// TIA Portal V17 program export: 1 tag tables, 1 data types, 3 data blocks, 11 code blocks (in call order from the OBs), 12 instance data blocks

VAR_GLOBAL   // PLC tag table "Default tag table"
   System_Byte AT %MB1 : Byte;
   FirstScan AT %M1.0 : Bool;
   DiagStatusUpdate AT %M1.1 : Bool;
   AlwaysTRUE AT %M1.2 : Bool;
   AlwaysFALSE AT %M1.3 : Bool;
   Clock_Byte AT %MB0 : Byte;
   Clock_10Hz AT %M0.0 : Bool;
   Clock_5Hz AT %M0.1 : Bool;
   "Clock_2.5Hz" AT %M0.2 : Bool;
   Clock_2Hz AT %M0.3 : Bool;
   "Clock_1.25Hz" AT %M0.4 : Bool;
   Clock_1Hz AT %M0.5 : Bool;
   "Clock_0.625Hz" AT %M0.6 : Bool;
   "Clock_0.5Hz" AT %M0.7 : Bool;
   MR_Pulse AT %Q4.0 : Bool;
   MA_Pulse AT %Q4.1 : Bool;
   MR_Direction AT %Q0.0 : Bool;
   MRenable AT %M2.0 : Bool;
   MRReset AT %M2.1 : Bool;
   MRHalt AT %M2.2 : Bool;
   "MRJog-" AT %M2.3 : Bool;
   "MRJog+" AT %M2.4 : Bool;
   MRMoveRelative AT %M2.5 : Bool;
   MRMoveAbsolute AT %M2.6 : Bool;
   MA_Direction AT %Q0.1 : Bool;
   MRPower AT %M2.7 : Bool;
   MRVelocity AT %M3.0 : Bool;
   MREnabled AT %M3.5 : Bool;
   MRHomed AT %M3.1 : Bool;
   MRMoveAbsDone AT %M3.2 : Bool;
   MRStandstill AT %M3.3 : Bool;
   MRError AT %M3.4 : Bool;
   MRActualVelocity AT %MD4 : Real;
   MRActualPosition AT %MD8 : Real;
   MS_Direction AT %Q0.2 : Bool;
   ME_Direction AT %Q0.3 : Bool;
   MS_Pulse AT %Q4.2 : Bool;
   ME_Pulse AT %Q4.3 : Bool;
   AUTOMATICO AT %M3.6 : Bool;
   MANUALE AT %M3.7 : Bool;
   RIPRISTINO AT %M12.0 : Bool;
   PASSO_RIP_01 AT %M12.1 : Bool;
   PASSO_RIP_02 AT %M12.2 : Bool;
   PASSO_RIP_03 AT %M12.3 : Bool;
   STARTCICLO AT %M12.6 : Bool;
   PASSO_CICLO_01 AT %M12.7 : Bool;
   PASSO_CICLO_03 AT %M13.0 : Bool;
   PASSO_CICLO_02 AT %M13.1 : Bool;
   MRSpQuotaMoveRel AT %MD14 : Real;
   MRSpVelocitaMoveRel AT %MD18 : Real;
   MRSpQuotaMoveAbs AT %MD22 : Real;
   MRSpVelocitaMoveAbs AT %MD26 : Real;
   AUX_OK AT %M12.4 : Bool;
   AUX_OK_T AT %M12.5 : Bool;
   RESET_ALLARMI AT %M13.2 : Bool;
   MR_MAN_RELATIVE AT %M13.3 : Bool;
   MR_MAN_ABSOLUTE AT %M13.4 : Bool;
   MR_MAN_HALT AT %M13.5 : Bool;
   MS_MAN_HALT AT %M13.6 : Bool;
   MS_MAN_RELATIVE AT %M13.7 : Bool;
   MS_MAN_ABSOLUTE AT %M30.0 : Bool;
   MA_MAN_HALT AT %M30.1 : Bool;
   MA_MAN_RELATIVE AT %M30.2 : Bool;
   MA_MAN_ABSOLUTE AT %M30.3 : Bool;
   ME_MAN_HALT AT %M30.4 : Bool;
   ME_MAN_RELATIVE AT %M30.5 : Bool;
   ME_MAN_ABSOLUTE AT %M30.6 : Bool;
   "E0.0 FC HOMING MS" AT %I0.0 : Bool;
   ALLA_01_FC_HOMING_MS AT %M30.7 : Bool;
   PASSO_PASSO AT %M31.0 : Bool;
   RIPRISTINATO AT %M31.1 : Bool;
   "E0.1 FC HOMING MR" AT %I0.1 : Bool;
   ALLA_02_FC_HOMING_MR AT %M31.2 : Bool;
END_VAR

TYPE "UDTMotori"
// stored: IsFailsafeCompliant false
   STRUCT
      pos : Struct
         "1" : Real;
         "2" : Real;
         "3" : Real;
         "4" : Real;
         "5" : Real;
      END_STRUCT;
      vel : Struct
         "1" : Real;
         "2" : Real;
         "3" : Real;
         "4" : Real;
         "5" : Real;
      END_STRUCT;
      acc : Struct
         "1" : Real;
         "2" : Real;
         "3" : Real;
         "4" : Real;
         "5" : Real;
      END_STRUCT;
      dec : Struct
         "1" : Real;
         "2" : Real;
         "3" : Real;
         "4" : Real;
         "5" : Real;
      END_STRUCT;
      IN : Struct
         Exe_MC_Reset : Bool;   // comando di reset
         En_MC_Power : Bool;   // abilitazione asse
         Exe_MC_Home : Bool;   // comando di homing
         Sp_Offset_Homing : Real;   // offset azzeramento
         Exe_MC_Halt : Bool;   // comando HALT
         Exe_Jog_Fwd : Bool;   // comando jog +
         Exe_Jog_Bkw : Bool;   // comando jog -
         Sp_Jog_Velocity : Real;   // set velocità JOG
         Exe_MC_Velocity : Bool;   // comando velocità
         Sp_MC_Velocity : Real;   // set velocità Move Velocity
         Exe_MC_MoveRelative : Bool;   // comando posizione relativa
         Sp_MoveRel_Distance : Real;   // set distanza Move Relative
         Sp_MoveRel_Velocity : Real;   // set velocità Move Relative
         Exe_MC_MoveAbs : Bool;   // comando posizione assoluta
         Sp_MoveAbs_Position : Real;   // set posizione Move Absolute
         Sp_MoveAbs_Velocity : Real;   // set velocità Move Absolute
         Exe_MC_ChangeDyna : Bool;   // comando cambio dinamica
         Sp_RampUpTime : Real;   // set tempo di rampa acc [s]
         Sp_RampDnTime : Real;   // set tempo di rampa dec [s]
      END_STRUCT;
      OUT : Struct
         Output_MC_Reset_Done : Bool;   // asse resettato
         Output_MC_AxisEnabled : Bool;   // asse abilitato
         Output_MC_AxisHomed : Bool;   // asse homed (referenziato)
         Output_MC_Halt_Done : Bool;   // asse in halt
         Output_MC_JogInVelocity : Bool;   // vel raggiunta
         Output_MC_MoveInVelocity : Bool;   // vel raggiunta
         Output_MC_MoveRel_Done : Bool;   // move realtive eseguito
         Output_MC_MoveAbs_Done : Bool;   // move absolute eseguito
         Output_MC_MoveAbs_Busy : Bool;   // move absolute in corso
         Output_MC_At_Standstill : Bool;   // asse fermo
         Output_MC_Error : Bool;   // asse in errore (or di vari bool)
         Output_ActVelocity : Real;   // velocity attuale (asse)
         Output_ActPos : Real;   // posizione attuale
      END_STRUCT;
   END_STRUCT;
END_TYPE

DATA_BLOCK "RICETTE"   // DB18
{ S7_Optimized_Access := 'TRUE' }
VERSION : 0.1
// stored: AutoNumber true, DBAccessibleFromOPCUA true, IsOnlyStoredInLoadMemory false, IsRetainMemResEnabled false, IsWriteProtectedInAS false, MemoryReserve 100
   VAR
      nomeRicetta : WString;
   END_VAR
BEGIN
END_DATA_BLOCK

DATA_BLOCK "DBParAssi"   // DB12
{ S7_Optimized_Access := 'TRUE' }
VERSION : 0.1
// stored: AutoNumber true, DBAccessibleFromOPCUA true, IsOnlyStoredInLoadMemory false, IsRetainMemResEnabled false, IsWriteProtectedInAS false, MemoryReserve 100
   VAR RETAIN
      MR : "UDTMotori";
      MA { S7_SetPoint := 'True'} : "UDTMotori";
      MS { S7_SetPoint := 'True'} : "UDTMotori";
      ME { S7_SetPoint := 'True'} : "UDTMotori";
   END_VAR
BEGIN
   MR.pos."1" := 120.0;   // [°] predisposizione (detorsione)
   MR.pos."2" := 10.0;   // [°] quota intermedia (detorsione parziale) / [°] quota intermedia
   MR.pos."3" := 0.0;   // [°] zero / [°]
   MR.pos."4" := 180.0;   // [°] ritorsione
   MR.vel."1" := 1000.0;   // [°/s] vel detorsione
   MR.vel."2" := 1000.0;   // [°/s] vel detorsione parziale
   MR.vel."3" := 200.0;   // [°/s] vel
   MR.vel."4" := 200.0;   // [°/s] vel ritorsione
   MR.IN.Sp_Jog_Velocity := 80.0;
   MR.IN.Sp_MoveRel_Velocity := 1000.0;
   MR.IN.Sp_MoveAbs_Velocity := 1000.0;
   MR.IN.Sp_RampUpTime := 2.0;
   MR.IN.Sp_RampDnTime := 2.0;
   MA.pos."1" := 7.5;   // [mm] quota detorsione / [mm]
   MA.pos."2" := 12.5;   // [mm] quota fissa era 12.5 / [mm]
   MA.pos."3" := 9.6;   // [mm] quota ritorsione / [mm]
   MA.pos."4" := 0.0;   // [mm]
   MA.IN.Sp_Jog_Velocity := 5.0;
   MA.IN.Sp_MoveRel_Velocity := 150.0;
   MA.IN.Sp_MoveAbs_Velocity := 50.0;
   MS.pos."1" := 220.0;   // [pulses] preset (800 0 giro completo) / [pulses] preset (400 0 giro completo)
   // MS.pos."2" : [pulses]
   MS.pos."3" := 95.0;   // [p] quota MA
   MS.vel."1" := 3000.0;   // [p/s]
   MS.vel."3" := 3000.0;   // [p/s]
   MS.IN.Sp_Jog_Velocity := 180.0;
   MS.IN.Sp_MoveRel_Distance := 230.0;
   MS.IN.Sp_MoveRel_Velocity := 1000.0;
   MS.IN.Sp_MoveAbs_Velocity := 1000.0;
   ME.pos."1" := 120.0;   // [°] quota blocco fili / [°]
   ME.pos."2" := 0.0;   // [°] Home position / [°]
   ME.IN.Sp_Jog_Velocity := 200.0;
   ME.IN.Sp_MoveRel_Velocity := 1000.0;
   ME.IN.Sp_MoveAbs_Velocity := 1000.0;
END_DATA_BLOCK

DATA_BLOCK "DB_ALLA"   // DB1
{ S7_Optimized_Access := 'FALSE' }
VERSION : 0.1
// stored: AutoNumber true, DBAccessibleFromOPCUA true, IsOnlyStoredInLoadMemory false, IsWriteProtectedInAS false
   VAR
      wordAlla01 : Word;
   END_VAR
BEGIN
END_DATA_BLOCK

ORGANIZATION_BLOCK "Main"   // OB1, LAD, ProgramCycle
TITLE = "Main Program Sweep (Cycle)"
{ S7_Optimized_Access := 'TRUE' }
VERSION : 0.1
// stored: AutoNumber true, IsIECCheckEnabled false, SetENOAutomatically false
   VAR_INPUT
      Initial_Call : Bool;   // Initial call of this OB
      Remanence : Bool;   // =True, if remanent data are available
   END_VAR
BEGIN

REGION Network 1 (SCL): FORZAMENTI

   //"E0.0 FC HOMING MS" := TRUE;
END_REGION

REGION Network 2 (SCL): LANCIO BLOCCHI

   "RESET_GENERALE"("FirstScan");
   "RESET_ALLA"("RESET_ALLARMI");


   "FB_STATI_MACCHINA_DB"();

   // CICLI
   "FB_RIPRISTINO_GEN_DB"();

   "FB_RIPRISTINO_MR_DB"();
   "FB_RIPRISTINO_MA_DB"();
   "FB_RIPRISTINO_MS_DB"();
   "FB_RIPRISTINO_ME_DB"();

   "FB_CICLO_DB"();

   "FB_ORG_ASSI_DB"();

   "ALLARMI_DB"();
END_REGION
END_ORGANIZATION_BLOCK

FUNCTION_BLOCK "FB_STATI_MACCHINA"   // FB2, LAD
{ S7_Optimized_Access := 'TRUE' }
VERSION : 0.1
// stored: AutoNumber true, IsIECCheckEnabled false, IsRetainMemResEnabled false, MemoryReserve 100, SetENOAutomatically false, UDAEnableTagReadback false
   VAR
      TAux { S7_SetPoint := 'True'} : TON_TIME;
      TResetAlla { S7_SetPoint := 'True'} : TON_TIME;
   END_VAR
BEGIN

REGION Network 1: AUX OK
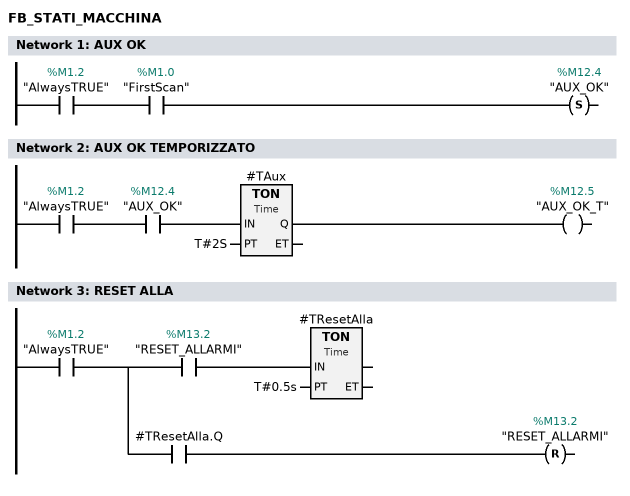
   RUNG wire#powerrail
      Contact( "AlwaysTRUE" )
      Contact( "FirstScan" )
      S_Coil( "AUX_OK" )
   END_RUNG
   // the same network as SCL:
   IF "AlwaysTRUE" AND "FirstScan" THEN "AUX_OK" := TRUE; END_IF;
END_REGION

REGION Network 2: AUX OK TEMPORIZZATO
   RUNG wire#powerrail
      Contact( "AlwaysTRUE" )
      Contact( "AUX_OK" )
      { S7_Templates := "time_type := Time" } #TAux.TON(pt := T#2S, et =>)
      Coil( "AUX_OK_T" )
   END_RUNG
   // the same network as SCL:
   #TAux(IN := "AlwaysTRUE" AND "AUX_OK", PT := T#2S);   // TON
   "AUX_OK_T" := #TAux.Q;
END_REGION

REGION Network 3: RESET ALLA
   RUNG wire#powerrail
      Contact( "AlwaysTRUE" )
      wire#w1
      Contact( "RESET_ALLARMI" )
      { S7_Templates := "time_type := Time" } #TResetAlla.TON(pt := T#0.5s, et =>)
   END_RUNG
   RUNG wire#w1
      Contact( #TResetAlla.Q )
      R_Coil( "RESET_ALLARMI" )
   END_RUNG
   // the same network as SCL:
   #TResetAlla(IN := "AlwaysTRUE" AND "RESET_ALLARMI", PT := T#0.5s);   // TON
   IF "AlwaysTRUE" AND #TResetAlla.Q THEN "RESET_ALLARMI" := FALSE; END_IF;
END_REGION

REGION Network 4 (SCL): MAN/AUTO

   "MANUALE" := NOT "AUTOMATICO";
END_REGION
END_FUNCTION_BLOCK

FUNCTION_BLOCK "FB_RIPRISTINO_GEN"
{ S7_Optimized_Access := 'TRUE' }
VERSION : 0.1
   VAR_OUTPUT 
      bDone : Bool;   // bDone
      fase : Int := 0;   // fase attiva
   END_VAR

   VAR_IN_OUT 
      bStart : Bool;   // start ciclo
   END_VAR

   VAR 
      condOkRipristino : Bool;
      T10 {InstructionName := 'TON_TIME'; LibVersion := '1.0'; S7_SetPoint := 'False'} : TON_TIME;
      T20 {InstructionName := 'TON_TIME'; LibVersion := '1.0'} : TON_TIME;
   END_VAR


BEGIN
	// ripristino generale
	
	#T10(IN := #fase = 10,
	     PT := t#1s);
	
	#T20(IN := #fase = 20,
	     PT := t#1s);
	
	// CONDIZIONI 
	// 
	#condOkRipristino := NOT "STARTCICLO" AND "AUX_OK_T";
	
	// reset start
	// 
	IF NOT #condOkRipristino THEN
	    "RIPRISTINO" := FALSE;
	END_IF;
	
	
	CASE #fase OF
	        
	    0: // attesa start ciclo
	        IF "RIPRISTINO" AND #condOkRipristino THEN
	            // comandi
	            // 
	            "FB_RIPRISTINO_MR_DB".bDone := FALSE;
	            "FB_RIPRISTINO_MA_DB".bDone := FALSE;
	            "FB_RIPRISTINO_MS_DB".bDone := FALSE;
	            "FB_RIPRISTINO_ME_DB".bDone := FALSE;
	            "RIPRISTINATO" := FALSE;
	            
	            "FB_RIPRISTINO_MA_DB".bStart := TRUE;
	            "FB_RIPRISTINO_ME_DB".bStart := TRUE;
	            
	            #fase := 10;
	        END_IF;
	        
	    10:
	        IF "FB_RIPRISTINO_MA_DB".bDone AND "FB_RIPRISTINO_ME_DB".bDone
	        THEN
	            // comandi 
	            // 
	            "FB_RIPRISTINO_MR_DB".bStart := TRUE;
	            "FB_RIPRISTINO_MS_DB".bStart := TRUE;
	            
	            #fase := 30;
	        END_IF;
	        
	    30: // fineciclo
	        IF   "FB_RIPRISTINO_MR_DB".bDone AND   "FB_RIPRISTINO_MS_DB".bDone        THEN
	            // comandi 
	            "RIPRISTINO" := FALSE;
	            "RIPRISTINATO" := TRUE;
	            #bDone := TRUE;
	            
	            #fase := 0;
	        END_IF;
	        
	END_CASE;
	
	
END_FUNCTION_BLOCK

FUNCTION_BLOCK "FB_ORG_ASSI"   // FB5, LAD
{ S7_Optimized_Access := 'TRUE' }
VERSION : 0.1
// stored: AutoNumber true, IsIECCheckEnabled false, IsRetainMemResEnabled false, MemoryReserve 100, SetENOAutomatically false, UDAEnableTagReadback false
   VAR
      CTRL_ASSE_STD_MA { S7_SetPoint := 'True'} : "CTRL_ASSE_STD";
      CTRL_ASSE_STD_MR { S7_SetPoint := 'True'} : "CTRL_ASSE_STD";
      CTRL_ASSE_STD_MS { S7_SetPoint := 'True'} : "CTRL_ASSE_STD";
      CTRL_ASSE_STD_ME { S7_SetPoint := 'True'} : "CTRL_ASSE_STD";
   END_VAR
BEGIN

REGION Network 1: RESET ALLARMI
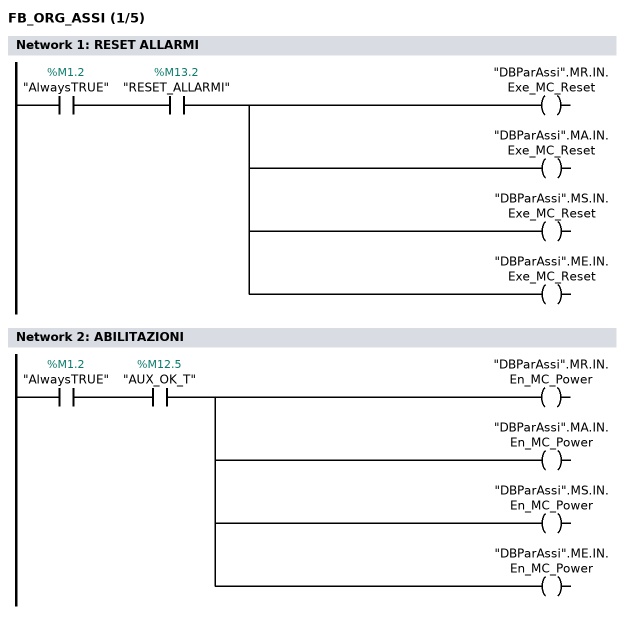
   RUNG wire#powerrail
      Contact( "AlwaysTRUE" )
      Contact( "RESET_ALLARMI" )
      wire#w1
      Coil( "DBParAssi".MR.IN.Exe_MC_Reset )
   END_RUNG
   RUNG wire#w1
      Coil( "DBParAssi".MA.IN.Exe_MC_Reset )
   END_RUNG
   RUNG wire#w1
      Coil( "DBParAssi".MS.IN.Exe_MC_Reset )
   END_RUNG
   RUNG wire#w1
      Coil( "DBParAssi".ME.IN.Exe_MC_Reset )
   END_RUNG
   // the same network as SCL:
   "DBParAssi".MR.IN.Exe_MC_Reset := "AlwaysTRUE" AND "RESET_ALLARMI";
   "DBParAssi".MA.IN.Exe_MC_Reset := "DBParAssi".MR.IN.Exe_MC_Reset;
   "DBParAssi".MS.IN.Exe_MC_Reset := "DBParAssi".MR.IN.Exe_MC_Reset;
   "DBParAssi".ME.IN.Exe_MC_Reset := "DBParAssi".MR.IN.Exe_MC_Reset;
END_REGION

REGION Network 2: ABILITAZIONI
   RUNG wire#powerrail
      Contact( "AlwaysTRUE" )
      Contact( "AUX_OK_T" )
      wire#w1
      Coil( "DBParAssi".MR.IN.En_MC_Power )
   END_RUNG
   RUNG wire#w1
      Coil( "DBParAssi".MA.IN.En_MC_Power )
   END_RUNG
   RUNG wire#w1
      Coil( "DBParAssi".MS.IN.En_MC_Power )
   END_RUNG
   RUNG wire#w1
      Coil( "DBParAssi".ME.IN.En_MC_Power )
   END_RUNG
   // the same network as SCL:
   "DBParAssi".MR.IN.En_MC_Power := "AlwaysTRUE" AND "AUX_OK_T";
   "DBParAssi".MA.IN.En_MC_Power := "DBParAssi".MR.IN.En_MC_Power;
   "DBParAssi".MS.IN.En_MC_Power := "DBParAssi".MR.IN.En_MC_Power;
   "DBParAssi".ME.IN.En_MC_Power := "DBParAssi".MR.IN.En_MC_Power;
END_REGION

REGION Network 3: ISTANZA MR
   // homing attivo = 3
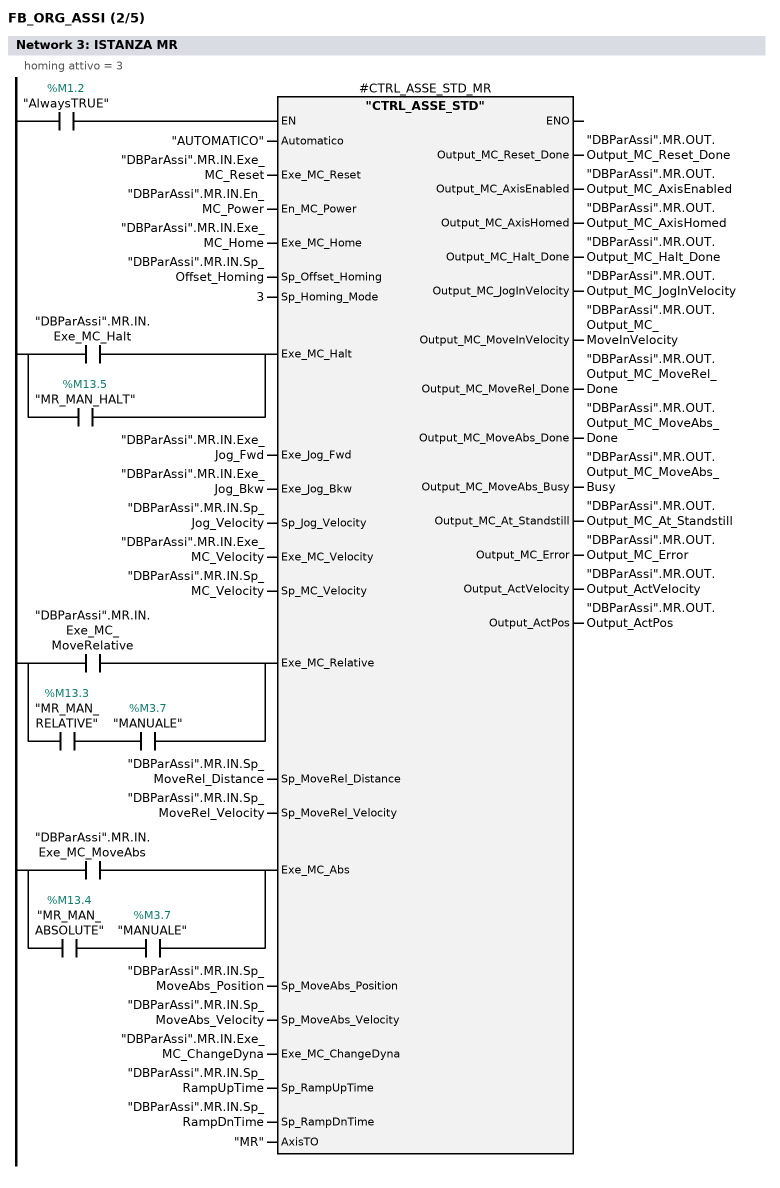
   RUNG wire#powerrail
      Contact( "AlwaysTRUE" )
      #CTRL_ASSE_STD_MR(Exe_MC_Halt := wire#w1, Exe_MC_Relative := wire#w2, Exe_MC_Abs := wire#w3, Automatico := "AUTOMATICO", Exe_MC_Reset := "DBParAssi".MR.IN.Exe_MC_Reset, En_MC_Power := "DBParAssi".MR.IN.En_MC_Power, Exe_MC_Home := "DBParAssi".MR.IN.Exe_MC_Home, Sp_Offset_Homing := "DBParAssi".MR.IN.Sp_Offset_Homing, Sp_Homing_Mode := 3, Exe_Jog_Fwd := "DBParAssi".MR.IN.Exe_Jog_Fwd, Exe_Jog_Bkw := "DBParAssi".MR.IN.Exe_Jog_Bkw, Sp_Jog_Velocity := "DBParAssi".MR.IN.Sp_Jog_Velocity, Exe_MC_Velocity := "DBParAssi".MR.IN.Exe_MC_Velocity, Sp_MC_Velocity := "DBParAssi".MR.IN.Sp_MC_Velocity, Sp_MoveRel_Distance := "DBParAssi".MR.IN.Sp_MoveRel_Distance, Sp_MoveRel_Velocity := "DBParAssi".MR.IN.Sp_MoveRel_Velocity, Sp_MoveAbs_Position := "DBParAssi".MR.IN.Sp_MoveAbs_Position, Sp_MoveAbs_Velocity := "DBParAssi".MR.IN.Sp_MoveAbs_Velocity, Exe_MC_ChangeDyna := "DBParAssi".MR.IN.Exe_MC_ChangeDyna, Sp_RampUpTime := "DBParAssi".MR.IN.Sp_RampUpTime, Sp_RampDnTime := "DBParAssi".MR.IN.Sp_RampDnTime, AxisTO := "MR", Output_MC_Reset_Done => "DBParAssi".MR.OUT.Output_MC_Reset_Done, Output_MC_AxisEnabled => "DBParAssi".MR.OUT.Output_MC_AxisEnabled, Output_MC_AxisHomed => "DBParAssi".MR.OUT.Output_MC_AxisHomed, Output_MC_Halt_Done => "DBParAssi".MR.OUT.Output_MC_Halt_Done, Output_MC_JogInVelocity => "DBParAssi".MR.OUT.Output_MC_JogInVelocity, Output_MC_MoveInVelocity => "DBParAssi".MR.OUT.Output_MC_MoveInVelocity, Output_MC_MoveRel_Done => "DBParAssi".MR.OUT.Output_MC_MoveRel_Done, Output_MC_MoveAbs_Done => "DBParAssi".MR.OUT.Output_MC_MoveAbs_Done, Output_MC_MoveAbs_Busy => "DBParAssi".MR.OUT.Output_MC_MoveAbs_Busy, Output_MC_At_Standstill => "DBParAssi".MR.OUT.Output_MC_At_Standstill, Output_MC_Error => "DBParAssi".MR.OUT.Output_MC_Error, Output_ActVelocity => "DBParAssi".MR.OUT.Output_ActVelocity, Output_ActPos => "DBParAssi".MR.OUT.Output_ActPos)
   END_RUNG
   RUNG wire#powerrail
      Contact( "DBParAssi".MR.IN.Exe_MC_Halt )
   END_RUNG wire#w1
   RUNG wire#powerrail
      Contact( "MR_MAN_HALT" )
   END_RUNG wire#w1
   RUNG wire#powerrail
      Contact( "DBParAssi".MR.IN.Exe_MC_MoveRelative )
   END_RUNG wire#w2
   RUNG wire#powerrail
      Contact( "MR_MAN_RELATIVE" )
      Contact( "MANUALE" )
   END_RUNG wire#w2
   RUNG wire#powerrail
      Contact( "DBParAssi".MR.IN.Exe_MC_MoveAbs )
   END_RUNG wire#w3
   RUNG wire#powerrail
      Contact( "MR_MAN_ABSOLUTE" )
      Contact( "MANUALE" )
   END_RUNG wire#w3
   // the same network as SCL:
   IF "AlwaysTRUE" THEN
       #CTRL_ASSE_STD_MR(Automatico := "AUTOMATICO",   // "CTRL_ASSE_STD"
                         Exe_MC_Reset := "DBParAssi".MR.IN.Exe_MC_Reset,
                         En_MC_Power := "DBParAssi".MR.IN.En_MC_Power,
                         Exe_MC_Home := "DBParAssi".MR.IN.Exe_MC_Home,
                         Sp_Offset_Homing := "DBParAssi".MR.IN.Sp_Offset_Homing,
                         Sp_Homing_Mode := 3,
                         Exe_MC_Halt := "DBParAssi".MR.IN.Exe_MC_Halt OR "MR_MAN_HALT",
                         Exe_Jog_Fwd := "DBParAssi".MR.IN.Exe_Jog_Fwd,
                         Exe_Jog_Bkw := "DBParAssi".MR.IN.Exe_Jog_Bkw,
                         Sp_Jog_Velocity := "DBParAssi".MR.IN.Sp_Jog_Velocity,
                         Exe_MC_Velocity := "DBParAssi".MR.IN.Exe_MC_Velocity,
                         Sp_MC_Velocity := "DBParAssi".MR.IN.Sp_MC_Velocity,
                         Exe_MC_Relative := "DBParAssi".MR.IN.Exe_MC_MoveRelative OR ("MR_MAN_RELATIVE" AND "MANUALE"),
                         Sp_MoveRel_Distance := "DBParAssi".MR.IN.Sp_MoveRel_Distance,
                         Sp_MoveRel_Velocity := "DBParAssi".MR.IN.Sp_MoveRel_Velocity,
                         Exe_MC_Abs := "DBParAssi".MR.IN.Exe_MC_MoveAbs OR ("MR_MAN_ABSOLUTE" AND "MANUALE"),
                         Sp_MoveAbs_Position := "DBParAssi".MR.IN.Sp_MoveAbs_Position,
                         Sp_MoveAbs_Velocity := "DBParAssi".MR.IN.Sp_MoveAbs_Velocity,
                         Exe_MC_ChangeDyna := "DBParAssi".MR.IN.Exe_MC_ChangeDyna,
                         Sp_RampUpTime := "DBParAssi".MR.IN.Sp_RampUpTime,
                         Sp_RampDnTime := "DBParAssi".MR.IN.Sp_RampDnTime,
                         AxisTO := "MR",
                         Output_MC_Reset_Done => "DBParAssi".MR.OUT.Output_MC_Reset_Done,
                         Output_MC_AxisEnabled => "DBParAssi".MR.OUT.Output_MC_AxisEnabled,
                         Output_MC_AxisHomed => "DBParAssi".MR.OUT.Output_MC_AxisHomed,
                         Output_MC_Halt_Done => "DBParAssi".MR.OUT.Output_MC_Halt_Done,
                         Output_MC_JogInVelocity => "DBParAssi".MR.OUT.Output_MC_JogInVelocity,
                         Output_MC_MoveInVelocity => "DBParAssi".MR.OUT.Output_MC_MoveInVelocity,
                         Output_MC_MoveRel_Done => "DBParAssi".MR.OUT.Output_MC_MoveRel_Done,
                         Output_MC_MoveAbs_Done => "DBParAssi".MR.OUT.Output_MC_MoveAbs_Done,
                         Output_MC_MoveAbs_Busy => "DBParAssi".MR.OUT.Output_MC_MoveAbs_Busy,
                         Output_MC_At_Standstill => "DBParAssi".MR.OUT.Output_MC_At_Standstill,
                         Output_MC_Error => "DBParAssi".MR.OUT.Output_MC_Error,
                         Output_ActVelocity => "DBParAssi".MR.OUT.Output_ActVelocity,
                         Output_ActPos => "DBParAssi".MR.OUT.Output_ActPos);
   END_IF;
END_REGION

REGION Network 4: ISTANZA MA
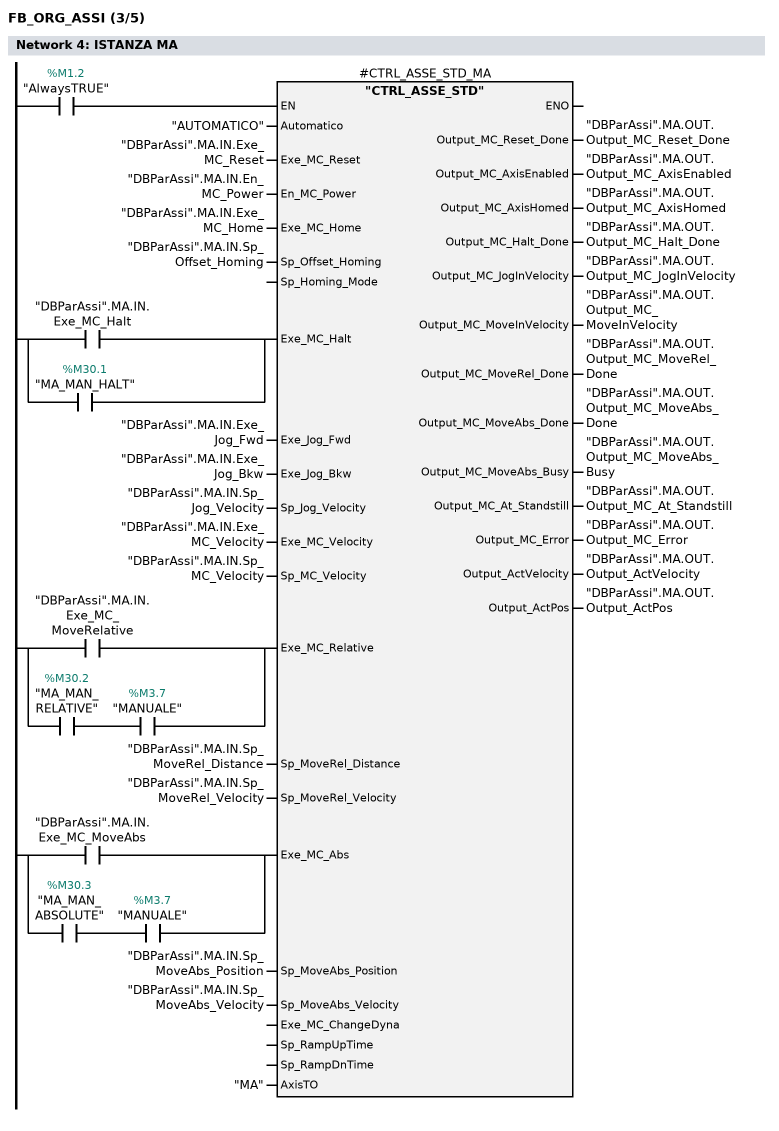
   RUNG wire#powerrail
      Contact( "AlwaysTRUE" )
      #CTRL_ASSE_STD_MA(Exe_MC_Halt := wire#w1, Exe_MC_Relative := wire#w2, Exe_MC_Abs := wire#w3, Automatico := "AUTOMATICO", Exe_MC_Reset := "DBParAssi".MA.IN.Exe_MC_Reset, En_MC_Power := "DBParAssi".MA.IN.En_MC_Power, Exe_MC_Home := "DBParAssi".MA.IN.Exe_MC_Home, Sp_Offset_Homing := "DBParAssi".MA.IN.Sp_Offset_Homing, Sp_Homing_Mode :=, Exe_Jog_Fwd := "DBParAssi".MA.IN.Exe_Jog_Fwd, Exe_Jog_Bkw := "DBParAssi".MA.IN.Exe_Jog_Bkw, Sp_Jog_Velocity := "DBParAssi".MA.IN.Sp_Jog_Velocity, Exe_MC_Velocity := "DBParAssi".MA.IN.Exe_MC_Velocity, Sp_MC_Velocity := "DBParAssi".MA.IN.Sp_MC_Velocity, Sp_MoveRel_Distance := "DBParAssi".MA.IN.Sp_MoveRel_Distance, Sp_MoveRel_Velocity := "DBParAssi".MA.IN.Sp_MoveRel_Velocity, Sp_MoveAbs_Position := "DBParAssi".MA.IN.Sp_MoveAbs_Position, Sp_MoveAbs_Velocity := "DBParAssi".MA.IN.Sp_MoveAbs_Velocity, Exe_MC_ChangeDyna :=, Sp_RampUpTime :=, Sp_RampDnTime :=, AxisTO := "MA", Output_MC_Reset_Done => "DBParAssi".MA.OUT.Output_MC_Reset_Done, Output_MC_AxisEnabled => "DBParAssi".MA.OUT.Output_MC_AxisEnabled, Output_MC_AxisHomed => "DBParAssi".MA.OUT.Output_MC_AxisHomed, Output_MC_Halt_Done => "DBParAssi".MA.OUT.Output_MC_Halt_Done, Output_MC_JogInVelocity => "DBParAssi".MA.OUT.Output_MC_JogInVelocity, Output_MC_MoveInVelocity => "DBParAssi".MA.OUT.Output_MC_MoveInVelocity, Output_MC_MoveRel_Done => "DBParAssi".MA.OUT.Output_MC_MoveRel_Done, Output_MC_MoveAbs_Done => "DBParAssi".MA.OUT.Output_MC_MoveAbs_Done, Output_MC_MoveAbs_Busy => "DBParAssi".MA.OUT.Output_MC_MoveAbs_Busy, Output_MC_At_Standstill => "DBParAssi".MA.OUT.Output_MC_At_Standstill, Output_MC_Error => "DBParAssi".MA.OUT.Output_MC_Error, Output_ActVelocity => "DBParAssi".MA.OUT.Output_ActVelocity, Output_ActPos => "DBParAssi".MA.OUT.Output_ActPos)
   END_RUNG
   RUNG wire#powerrail
      Contact( "DBParAssi".MA.IN.Exe_MC_Halt )
   END_RUNG wire#w1
   RUNG wire#powerrail
      Contact( "MA_MAN_HALT" )
   END_RUNG wire#w1
   RUNG wire#powerrail
      Contact( "DBParAssi".MA.IN.Exe_MC_MoveRelative )
   END_RUNG wire#w2
   RUNG wire#powerrail
      Contact( "MA_MAN_RELATIVE" )
      Contact( "MANUALE" )
   END_RUNG wire#w2
   RUNG wire#powerrail
      Contact( "DBParAssi".MA.IN.Exe_MC_MoveAbs )
   END_RUNG wire#w3
   RUNG wire#powerrail
      Contact( "MA_MAN_ABSOLUTE" )
      Contact( "MANUALE" )
   END_RUNG wire#w3
   // the same network as SCL:
   IF "AlwaysTRUE" THEN
       #CTRL_ASSE_STD_MA(Automatico := "AUTOMATICO",   // "CTRL_ASSE_STD"
                         Exe_MC_Reset := "DBParAssi".MA.IN.Exe_MC_Reset,
                         En_MC_Power := "DBParAssi".MA.IN.En_MC_Power,
                         Exe_MC_Home := "DBParAssi".MA.IN.Exe_MC_Home,
                         Sp_Offset_Homing := "DBParAssi".MA.IN.Sp_Offset_Homing,
                         Exe_MC_Halt := "DBParAssi".MA.IN.Exe_MC_Halt OR "MA_MAN_HALT",
                         Exe_Jog_Fwd := "DBParAssi".MA.IN.Exe_Jog_Fwd,
                         Exe_Jog_Bkw := "DBParAssi".MA.IN.Exe_Jog_Bkw,
                         Sp_Jog_Velocity := "DBParAssi".MA.IN.Sp_Jog_Velocity,
                         Exe_MC_Velocity := "DBParAssi".MA.IN.Exe_MC_Velocity,
                         Sp_MC_Velocity := "DBParAssi".MA.IN.Sp_MC_Velocity,
                         Exe_MC_Relative := "DBParAssi".MA.IN.Exe_MC_MoveRelative OR ("MA_MAN_RELATIVE" AND "MANUALE"),
                         Sp_MoveRel_Distance := "DBParAssi".MA.IN.Sp_MoveRel_Distance,
                         Sp_MoveRel_Velocity := "DBParAssi".MA.IN.Sp_MoveRel_Velocity,
                         Exe_MC_Abs := "DBParAssi".MA.IN.Exe_MC_MoveAbs OR ("MA_MAN_ABSOLUTE" AND "MANUALE"),
                         Sp_MoveAbs_Position := "DBParAssi".MA.IN.Sp_MoveAbs_Position,
                         Sp_MoveAbs_Velocity := "DBParAssi".MA.IN.Sp_MoveAbs_Velocity,
                         AxisTO := "MA",
                         Output_MC_Reset_Done => "DBParAssi".MA.OUT.Output_MC_Reset_Done,
                         Output_MC_AxisEnabled => "DBParAssi".MA.OUT.Output_MC_AxisEnabled,
                         Output_MC_AxisHomed => "DBParAssi".MA.OUT.Output_MC_AxisHomed,
                         Output_MC_Halt_Done => "DBParAssi".MA.OUT.Output_MC_Halt_Done,
                         Output_MC_JogInVelocity => "DBParAssi".MA.OUT.Output_MC_JogInVelocity,
                         Output_MC_MoveInVelocity => "DBParAssi".MA.OUT.Output_MC_MoveInVelocity,
                         Output_MC_MoveRel_Done => "DBParAssi".MA.OUT.Output_MC_MoveRel_Done,
                         Output_MC_MoveAbs_Done => "DBParAssi".MA.OUT.Output_MC_MoveAbs_Done,
                         Output_MC_MoveAbs_Busy => "DBParAssi".MA.OUT.Output_MC_MoveAbs_Busy,
                         Output_MC_At_Standstill => "DBParAssi".MA.OUT.Output_MC_At_Standstill,
                         Output_MC_Error => "DBParAssi".MA.OUT.Output_MC_Error,
                         Output_ActVelocity => "DBParAssi".MA.OUT.Output_ActVelocity,
                         Output_ActPos => "DBParAssi".MA.OUT.Output_ActPos);
   END_IF;
END_REGION

REGION Network 5 (SCL): ISTANZA MA SCL

   // #CTRL_ASSE_STD_MA(Exe_MC_Reset:="DBParAssi".MA.IN.Exe_MC_Reset,
   //                         En_MC_Power:="DBParAssi".MA.IN.En_MC_Power,
   //                         Exe_MC_Home:="DBParAssi".MA.IN.Exe_MC_Home,
   //                         Sp_Offset_Homing:="DBParAssi".MA.IN.Sp_Offset_Homing,
   //                         Exe_MC_Halt:="DBParAssi".MA.IN.Exe_MC_Halt,
   //                         Exe_Jog_Fwd:="DBParAssi".MA.IN.Exe_Jog_Fwd,
   //                         Exe_Jog_Bkw:="DBParAssi".MA.IN.Exe_Jog_Bkw,
   //                         Sp_Jog_Velocity:="DBParAssi".MA.IN.Sp_Jog_Velocity,
   //                         Exe_MC_Velocity:="DBParAssi".MA.IN.Exe_MC_Velocity,
   //                         Sp_MC_Velocity:="DBParAssi".MA.IN.Sp_MC_Velocity,
   //                         Exe_MC_Relative:="DBParAssi".MA.IN.Exe_MC_MoveRelative,
   //                         Sp_MoveRel_Distance:="DBParAssi".MA.IN.Sp_MoveRel_Distance,
   //                         Sp_MoveRel_Velocity:="DBParAssi".MA.IN.Sp_MoveRel_Velocity,
   //                         Exe_MC_Abs:="DBParAssi".MA.IN.Exe_MC_MoveAbs,
   //                         Sp_MoveAbs_Position:="DBParAssi".MA.IN.Sp_MoveAbs_Position,
   //                         Sp_MoveAbs_Velocity:="DBParAssi".MA.IN.Sp_MoveAbs_Velocity,
   //                         Output_MC_Reset_Done=>"DBParAssi".MA.OUT.Output_MC_Reset_Done,
   //                         Output_MC_AxisEnabled=>"DBParAssi".MA.OUT.Output_MC_AxisEnabled,
   //                         Output_MC_AxisHomed=>"DBParAssi".MA.OUT.Output_MC_AxisHomed,
   //                         Output_MC_Halt_Done=>"DBParAssi".MA.OUT.Output_MC_Halt_Done,
   //                         Output_MC_JogInVelocity=>"DBParAssi".MA.OUT.Output_MC_Reset_Done,
   //                         Output_MC_MoveInVelocity=>"DBParAssi".MA.OUT.Output_MC_MoveInVelocity,
   //                         Output_MC_MoveRel_Done=>"DBParAssi".MA.OUT.Output_MC_MoveRel_Done,
   //                         Output_MC_MoveAbs_Done=>"DBParAssi".MA.OUT.Output_MC_MoveAbs_Done,
   //                         Output_MC_MoveAbs_Busy=>"DBParAssi".MA.OUT.Output_MC_MoveAbs_Busy,
   //                         Output_MC_At_Standstill=>"DBParAssi".MA.OUT.Output_MC_Reset_Done,
   //                         Output_MC_Error=>"DBParAssi".MA.OUT.Output_MC_Error,
   //                         Output_ActVelocity=>"DBParAssi".MA.OUT.Output_ActVelocity,
   //                         Output_ActPos=>"DBParAssi".MA.OUT.Output_ActPos,
   //                         AxisTO:="MA");
END_REGION

REGION Network 6: ISTANZA MS
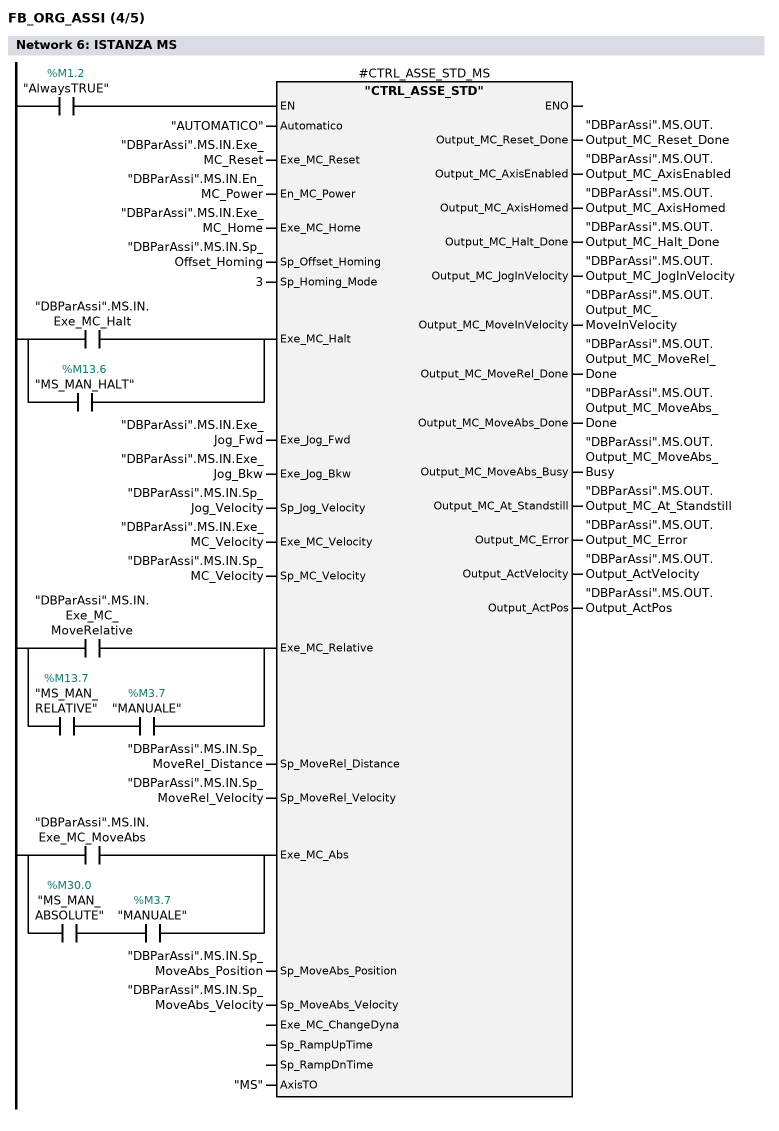
   RUNG wire#powerrail
      Contact( "AlwaysTRUE" )
      #CTRL_ASSE_STD_MS(Exe_MC_Halt := wire#w1, Exe_MC_Relative := wire#w2, Exe_MC_Abs := wire#w3, Automatico := "AUTOMATICO", Exe_MC_Reset := "DBParAssi".MS.IN.Exe_MC_Reset, En_MC_Power := "DBParAssi".MS.IN.En_MC_Power, Exe_MC_Home := "DBParAssi".MS.IN.Exe_MC_Home, Sp_Offset_Homing := "DBParAssi".MS.IN.Sp_Offset_Homing, Sp_Homing_Mode := 3, Exe_Jog_Fwd := "DBParAssi".MS.IN.Exe_Jog_Fwd, Exe_Jog_Bkw := "DBParAssi".MS.IN.Exe_Jog_Bkw, Sp_Jog_Velocity := "DBParAssi".MS.IN.Sp_Jog_Velocity, Exe_MC_Velocity := "DBParAssi".MS.IN.Exe_MC_Velocity, Sp_MC_Velocity := "DBParAssi".MS.IN.Sp_MC_Velocity, Sp_MoveRel_Distance := "DBParAssi".MS.IN.Sp_MoveRel_Distance, Sp_MoveRel_Velocity := "DBParAssi".MS.IN.Sp_MoveRel_Velocity, Sp_MoveAbs_Position := "DBParAssi".MS.IN.Sp_MoveAbs_Position, Sp_MoveAbs_Velocity := "DBParAssi".MS.IN.Sp_MoveAbs_Velocity, Exe_MC_ChangeDyna :=, Sp_RampUpTime :=, Sp_RampDnTime :=, AxisTO := "MS", Output_MC_Reset_Done => "DBParAssi".MS.OUT.Output_MC_Reset_Done, Output_MC_AxisEnabled => "DBParAssi".MS.OUT.Output_MC_AxisEnabled, Output_MC_AxisHomed => "DBParAssi".MS.OUT.Output_MC_AxisHomed, Output_MC_Halt_Done => "DBParAssi".MS.OUT.Output_MC_Halt_Done, Output_MC_JogInVelocity => "DBParAssi".MS.OUT.Output_MC_JogInVelocity, Output_MC_MoveInVelocity => "DBParAssi".MS.OUT.Output_MC_MoveInVelocity, Output_MC_MoveRel_Done => "DBParAssi".MS.OUT.Output_MC_MoveRel_Done, Output_MC_MoveAbs_Done => "DBParAssi".MS.OUT.Output_MC_MoveAbs_Done, Output_MC_MoveAbs_Busy => "DBParAssi".MS.OUT.Output_MC_MoveAbs_Busy, Output_MC_At_Standstill => "DBParAssi".MS.OUT.Output_MC_At_Standstill, Output_MC_Error => "DBParAssi".MS.OUT.Output_MC_Error, Output_ActVelocity => "DBParAssi".MS.OUT.Output_ActVelocity, Output_ActPos => "DBParAssi".MS.OUT.Output_ActPos)
   END_RUNG
   RUNG wire#powerrail
      Contact( "DBParAssi".MS.IN.Exe_MC_Halt )
   END_RUNG wire#w1
   RUNG wire#powerrail
      Contact( "MS_MAN_HALT" )
   END_RUNG wire#w1
   RUNG wire#powerrail
      Contact( "DBParAssi".MS.IN.Exe_MC_MoveRelative )
   END_RUNG wire#w2
   RUNG wire#powerrail
      Contact( "MS_MAN_RELATIVE" )
      Contact( "MANUALE" )
   END_RUNG wire#w2
   RUNG wire#powerrail
      Contact( "DBParAssi".MS.IN.Exe_MC_MoveAbs )
   END_RUNG wire#w3
   RUNG wire#powerrail
      Contact( "MS_MAN_ABSOLUTE" )
      Contact( "MANUALE" )
   END_RUNG wire#w3
   // the same network as SCL:
   IF "AlwaysTRUE" THEN
       #CTRL_ASSE_STD_MS(Automatico := "AUTOMATICO",   // "CTRL_ASSE_STD"
                         Exe_MC_Reset := "DBParAssi".MS.IN.Exe_MC_Reset,
                         En_MC_Power := "DBParAssi".MS.IN.En_MC_Power,
                         Exe_MC_Home := "DBParAssi".MS.IN.Exe_MC_Home,
                         Sp_Offset_Homing := "DBParAssi".MS.IN.Sp_Offset_Homing,
                         Sp_Homing_Mode := 3,
                         Exe_MC_Halt := "DBParAssi".MS.IN.Exe_MC_Halt OR "MS_MAN_HALT",
                         Exe_Jog_Fwd := "DBParAssi".MS.IN.Exe_Jog_Fwd,
                         Exe_Jog_Bkw := "DBParAssi".MS.IN.Exe_Jog_Bkw,
                         Sp_Jog_Velocity := "DBParAssi".MS.IN.Sp_Jog_Velocity,
                         Exe_MC_Velocity := "DBParAssi".MS.IN.Exe_MC_Velocity,
                         Sp_MC_Velocity := "DBParAssi".MS.IN.Sp_MC_Velocity,
                         Exe_MC_Relative := "DBParAssi".MS.IN.Exe_MC_MoveRelative OR ("MS_MAN_RELATIVE" AND "MANUALE"),
                         Sp_MoveRel_Distance := "DBParAssi".MS.IN.Sp_MoveRel_Distance,
                         Sp_MoveRel_Velocity := "DBParAssi".MS.IN.Sp_MoveRel_Velocity,
                         Exe_MC_Abs := "DBParAssi".MS.IN.Exe_MC_MoveAbs OR ("MS_MAN_ABSOLUTE" AND "MANUALE"),
                         Sp_MoveAbs_Position := "DBParAssi".MS.IN.Sp_MoveAbs_Position,
                         Sp_MoveAbs_Velocity := "DBParAssi".MS.IN.Sp_MoveAbs_Velocity,
                         AxisTO := "MS",
                         Output_MC_Reset_Done => "DBParAssi".MS.OUT.Output_MC_Reset_Done,
                         Output_MC_AxisEnabled => "DBParAssi".MS.OUT.Output_MC_AxisEnabled,
                         Output_MC_AxisHomed => "DBParAssi".MS.OUT.Output_MC_AxisHomed,
                         Output_MC_Halt_Done => "DBParAssi".MS.OUT.Output_MC_Halt_Done,
                         Output_MC_JogInVelocity => "DBParAssi".MS.OUT.Output_MC_JogInVelocity,
                         Output_MC_MoveInVelocity => "DBParAssi".MS.OUT.Output_MC_MoveInVelocity,
                         Output_MC_MoveRel_Done => "DBParAssi".MS.OUT.Output_MC_MoveRel_Done,
                         Output_MC_MoveAbs_Done => "DBParAssi".MS.OUT.Output_MC_MoveAbs_Done,
                         Output_MC_MoveAbs_Busy => "DBParAssi".MS.OUT.Output_MC_MoveAbs_Busy,
                         Output_MC_At_Standstill => "DBParAssi".MS.OUT.Output_MC_At_Standstill,
                         Output_MC_Error => "DBParAssi".MS.OUT.Output_MC_Error,
                         Output_ActVelocity => "DBParAssi".MS.OUT.Output_ActVelocity,
                         Output_ActPos => "DBParAssi".MS.OUT.Output_ActPos);
   END_IF;
END_REGION

REGION Network 7: ISTANZA ME
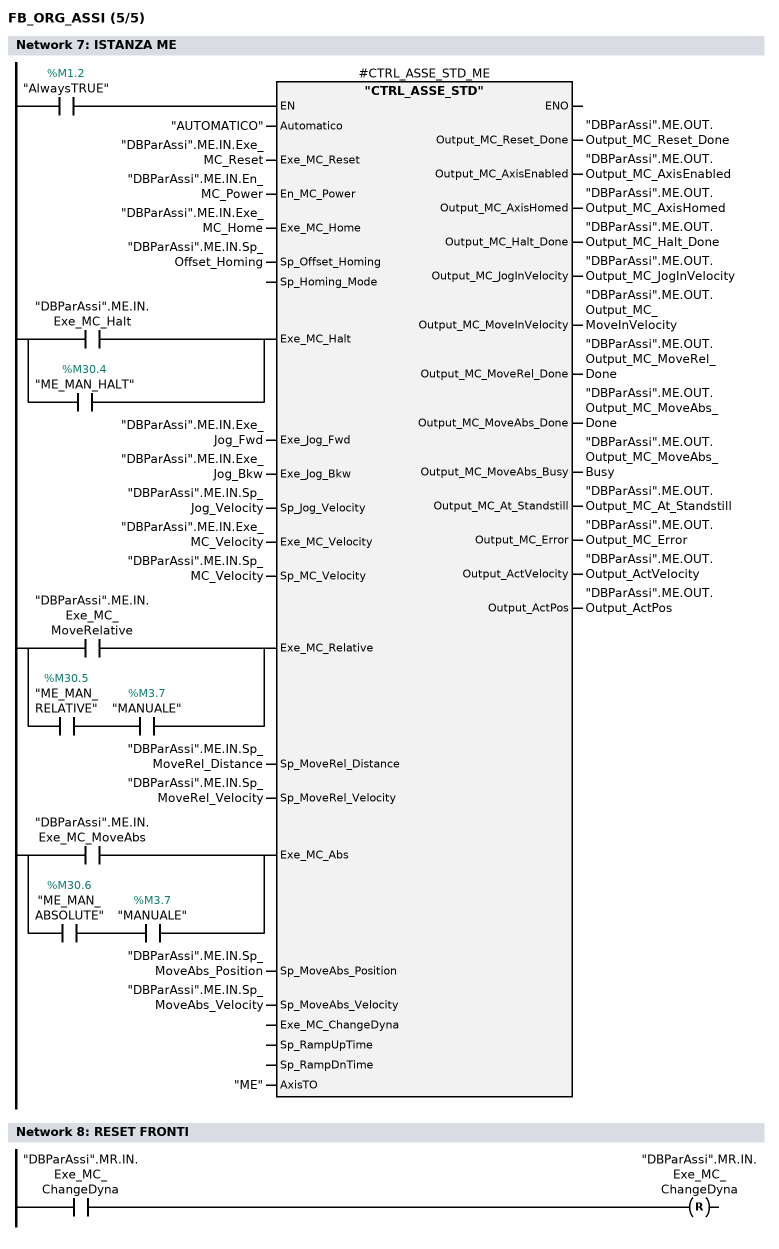
   RUNG wire#powerrail
      Contact( "AlwaysTRUE" )
      #CTRL_ASSE_STD_ME(Exe_MC_Halt := wire#w1, Exe_MC_Relative := wire#w2, Exe_MC_Abs := wire#w3, Automatico := "AUTOMATICO", Exe_MC_Reset := "DBParAssi".ME.IN.Exe_MC_Reset, En_MC_Power := "DBParAssi".ME.IN.En_MC_Power, Exe_MC_Home := "DBParAssi".ME.IN.Exe_MC_Home, Sp_Offset_Homing := "DBParAssi".ME.IN.Sp_Offset_Homing, Sp_Homing_Mode :=, Exe_Jog_Fwd := "DBParAssi".ME.IN.Exe_Jog_Fwd, Exe_Jog_Bkw := "DBParAssi".ME.IN.Exe_Jog_Bkw, Sp_Jog_Velocity := "DBParAssi".ME.IN.Sp_Jog_Velocity, Exe_MC_Velocity := "DBParAssi".ME.IN.Exe_MC_Velocity, Sp_MC_Velocity := "DBParAssi".ME.IN.Sp_MC_Velocity, Sp_MoveRel_Distance := "DBParAssi".ME.IN.Sp_MoveRel_Distance, Sp_MoveRel_Velocity := "DBParAssi".ME.IN.Sp_MoveRel_Velocity, Sp_MoveAbs_Position := "DBParAssi".ME.IN.Sp_MoveAbs_Position, Sp_MoveAbs_Velocity := "DBParAssi".ME.IN.Sp_MoveAbs_Velocity, Exe_MC_ChangeDyna :=, Sp_RampUpTime :=, Sp_RampDnTime :=, AxisTO := "ME", Output_MC_Reset_Done => "DBParAssi".ME.OUT.Output_MC_Reset_Done, Output_MC_AxisEnabled => "DBParAssi".ME.OUT.Output_MC_AxisEnabled, Output_MC_AxisHomed => "DBParAssi".ME.OUT.Output_MC_AxisHomed, Output_MC_Halt_Done => "DBParAssi".ME.OUT.Output_MC_Halt_Done, Output_MC_JogInVelocity => "DBParAssi".ME.OUT.Output_MC_JogInVelocity, Output_MC_MoveInVelocity => "DBParAssi".ME.OUT.Output_MC_MoveInVelocity, Output_MC_MoveRel_Done => "DBParAssi".ME.OUT.Output_MC_MoveRel_Done, Output_MC_MoveAbs_Done => "DBParAssi".ME.OUT.Output_MC_MoveAbs_Done, Output_MC_MoveAbs_Busy => "DBParAssi".ME.OUT.Output_MC_MoveAbs_Busy, Output_MC_At_Standstill => "DBParAssi".ME.OUT.Output_MC_At_Standstill, Output_MC_Error => "DBParAssi".ME.OUT.Output_MC_Error, Output_ActVelocity => "DBParAssi".ME.OUT.Output_ActVelocity, Output_ActPos => "DBParAssi".ME.OUT.Output_ActPos)
   END_RUNG
   RUNG wire#powerrail
      Contact( "DBParAssi".ME.IN.Exe_MC_Halt )
   END_RUNG wire#w1
   RUNG wire#powerrail
      Contact( "ME_MAN_HALT" )
   END_RUNG wire#w1
   RUNG wire#powerrail
      Contact( "DBParAssi".ME.IN.Exe_MC_MoveRelative )
   END_RUNG wire#w2
   RUNG wire#powerrail
      Contact( "ME_MAN_RELATIVE" )
      Contact( "MANUALE" )
   END_RUNG wire#w2
   RUNG wire#powerrail
      Contact( "DBParAssi".ME.IN.Exe_MC_MoveAbs )
   END_RUNG wire#w3
   RUNG wire#powerrail
      Contact( "ME_MAN_ABSOLUTE" )
      Contact( "MANUALE" )
   END_RUNG wire#w3
   // the same network as SCL:
   IF "AlwaysTRUE" THEN
       #CTRL_ASSE_STD_ME(Automatico := "AUTOMATICO",   // "CTRL_ASSE_STD"
                         Exe_MC_Reset := "DBParAssi".ME.IN.Exe_MC_Reset,
                         En_MC_Power := "DBParAssi".ME.IN.En_MC_Power,
                         Exe_MC_Home := "DBParAssi".ME.IN.Exe_MC_Home,
                         Sp_Offset_Homing := "DBParAssi".ME.IN.Sp_Offset_Homing,
                         Exe_MC_Halt := "DBParAssi".ME.IN.Exe_MC_Halt OR "ME_MAN_HALT",
                         Exe_Jog_Fwd := "DBParAssi".ME.IN.Exe_Jog_Fwd,
                         Exe_Jog_Bkw := "DBParAssi".ME.IN.Exe_Jog_Bkw,
                         Sp_Jog_Velocity := "DBParAssi".ME.IN.Sp_Jog_Velocity,
                         Exe_MC_Velocity := "DBParAssi".ME.IN.Exe_MC_Velocity,
                         Sp_MC_Velocity := "DBParAssi".ME.IN.Sp_MC_Velocity,
                         Exe_MC_Relative := "DBParAssi".ME.IN.Exe_MC_MoveRelative OR ("ME_MAN_RELATIVE" AND "MANUALE"),
                         Sp_MoveRel_Distance := "DBParAssi".ME.IN.Sp_MoveRel_Distance,
                         Sp_MoveRel_Velocity := "DBParAssi".ME.IN.Sp_MoveRel_Velocity,
                         Exe_MC_Abs := "DBParAssi".ME.IN.Exe_MC_MoveAbs OR ("ME_MAN_ABSOLUTE" AND "MANUALE"),
                         Sp_MoveAbs_Position := "DBParAssi".ME.IN.Sp_MoveAbs_Position,
                         Sp_MoveAbs_Velocity := "DBParAssi".ME.IN.Sp_MoveAbs_Velocity,
                         AxisTO := "ME",
                         Output_MC_Reset_Done => "DBParAssi".ME.OUT.Output_MC_Reset_Done,
                         Output_MC_AxisEnabled => "DBParAssi".ME.OUT.Output_MC_AxisEnabled,
                         Output_MC_AxisHomed => "DBParAssi".ME.OUT.Output_MC_AxisHomed,
                         Output_MC_Halt_Done => "DBParAssi".ME.OUT.Output_MC_Halt_Done,
                         Output_MC_JogInVelocity => "DBParAssi".ME.OUT.Output_MC_JogInVelocity,
                         Output_MC_MoveInVelocity => "DBParAssi".ME.OUT.Output_MC_MoveInVelocity,
                         Output_MC_MoveRel_Done => "DBParAssi".ME.OUT.Output_MC_MoveRel_Done,
                         Output_MC_MoveAbs_Done => "DBParAssi".ME.OUT.Output_MC_MoveAbs_Done,
                         Output_MC_MoveAbs_Busy => "DBParAssi".ME.OUT.Output_MC_MoveAbs_Busy,
                         Output_MC_At_Standstill => "DBParAssi".ME.OUT.Output_MC_At_Standstill,
                         Output_MC_Error => "DBParAssi".ME.OUT.Output_MC_Error,
                         Output_ActVelocity => "DBParAssi".ME.OUT.Output_ActVelocity,
                         Output_ActPos => "DBParAssi".ME.OUT.Output_ActPos);
   END_IF;
END_REGION

REGION Network 8: RESET FRONTI
   RUNG wire#powerrail
      Contact( "DBParAssi".MR.IN.Exe_MC_ChangeDyna )
      R_Coil( "DBParAssi".MR.IN.Exe_MC_ChangeDyna )
   END_RUNG
   // the same network as SCL:
   IF "DBParAssi".MR.IN.Exe_MC_ChangeDyna THEN "DBParAssi".MR.IN.Exe_MC_ChangeDyna := FALSE; END_IF;
END_REGION
END_FUNCTION_BLOCK

FUNCTION_BLOCK "ALLARMI"   // FB13, LAD
TITLE = COMPILAZIONE ALLARMI HMI
{ S7_Optimized_Access := 'TRUE' }
VERSION : 0.1
// stored: AutoNumber true, IsIECCheckEnabled false, IsRetainMemResEnabled false, MemoryReserve 100, SetENOAutomatically false, UDAEnableTagReadback false
BEGIN

REGION Network 1: ALLA HOMING MS
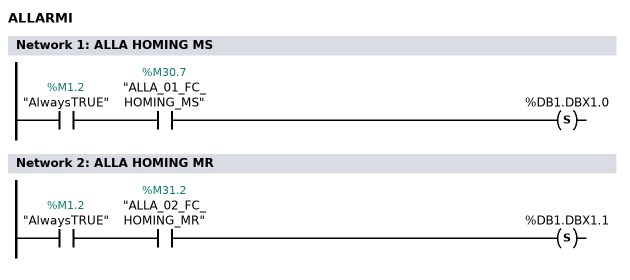
   RUNG wire#powerrail
      Contact( "AlwaysTRUE" )
      Contact( "ALLA_01_FC_HOMING_MS" )
      S_Coil( %DB1.DBX1.0 )
   END_RUNG
   // the same network as SCL:
   IF "AlwaysTRUE" AND "ALLA_01_FC_HOMING_MS" THEN %DB1.DBX1.0 := TRUE; END_IF;
END_REGION

REGION Network 2: ALLA HOMING MR
   RUNG wire#powerrail
      Contact( "AlwaysTRUE" )
      Contact( "ALLA_02_FC_HOMING_MR" )
      S_Coil( %DB1.DBX1.1 )
   END_RUNG
   // the same network as SCL:
   IF "AlwaysTRUE" AND "ALLA_02_FC_HOMING_MR" THEN %DB1.DBX1.1 := TRUE; END_IF;
END_REGION
END_FUNCTION_BLOCK

ORGANIZATION_BLOCK "Startup"
TITLE = "Complete Restart"
{ S7_Optimized_Access := 'TRUE' }
VERSION : 0.1

BEGIN
	
	// STATI
	"AUTOMATICO" := TRUE;
	"MANUALE" := FALSE;
	
	"FB_RIPRISTINO_GEN_DB".fase := 0;
	"FB_RIPRISTINO_GEN_DB".bDone := 0;
	
	"FB_RIPRISTINO_MR_DB".fase := 0;
	"FB_RIPRISTINO_MR_DB".bDone := 0;
	"FB_RIPRISTINO_MA_DB".fase := 0;
	"FB_RIPRISTINO_MA_DB".bDone := 0;
	"FB_RIPRISTINO_MS_DB".fase := 0;
	"FB_RIPRISTINO_MS_DB".bDone := 0;
	"FB_RIPRISTINO_ME_DB".fase := 0;
	"FB_RIPRISTINO_ME_DB".bDone := 0;
	
	"PASSO_PASSO" := 0;
	
	"FB_CICLO_DB".fase := 0;
	
	// forzamento ripristino
	"RIPRISTINO" := true;
	
	// forzamento valori e fronte per acce/dece
	// "DBParAssi".MR.IN.Sp_RampDnTime := 1.0;
	// "DBParAssi".MR.IN.Sp_RampUpTime := 1.0;
	// "DBParAssi".MR.IN.Exe_MC_ChangeDyna := TRUE;
	// 
	
	
	// Ricetta di default
	// 
	"RICETTE".nomeRicetta:=WSTRING#'Filo 1 ok';
	
	
END_ORGANIZATION_BLOCK

FUNCTION "RESET_ALLA" : Void
{ S7_Optimized_Access := 'TRUE' }
VERSION : 0.1
   VAR_INPUT 
      trigger : Bool;
   END_VAR


BEGIN
	// reset allarmi
	// 
	
	IF #trigger THEN
	    // reset alla homing
	    "ALLA_01_FC_HOMING_MS" := FALSE;
	    "ALLA_02_FC_HOMING_MR" := FALSE;
	    "FB_RIPRISTINO_GEN_DB".fase := 0;
	    "FB_RIPRISTINO_MR_DB".fase := 0;
	    "FB_RIPRISTINO_MS_DB".fase := 0;
	    
	// DB ALLARMI    
	    "DB_ALLA".wordAlla01 := 0;
	    
	END_IF;
	
END_FUNCTION

FUNCTION "RESET_GENERALE" : Void
{ S7_Optimized_Access := 'TRUE' }
VERSION : 0.1
   VAR_INPUT 
      trigger : Bool;
   END_VAR


BEGIN
	// reset generale
	// 
	IF #trigger OR "RESET_ALLARMI" THEN
	    "DBParAssi".MR.IN.Exe_MC_MoveRelative := FALSE;
	    "DBParAssi".MR.IN.Exe_MC_MoveAbs := FALSE;
	    "DBParAssi".MR.IN.Exe_MC_Halt := FALSE;
	    "FB_RIPRISTINO_MR_DB".bStart := 0;
	    "FB_RIPRISTINO_MR_DB".fase := 0;
	    "FB_RIPRISTINO_MR_DB".bDone := 0;
	    
	    "DBParAssi".MA.IN.Exe_MC_MoveRelative := FALSE;
	    "DBParAssi".MA.IN.Exe_MC_MoveAbs := FALSE;
	    "DBParAssi".MA.IN.Exe_MC_Halt := FALSE;
	    "FB_RIPRISTINO_MA_DB".bStart := 0;
	    "FB_RIPRISTINO_MA_DB".fase := 0;
	    "FB_RIPRISTINO_MA_DB".bDone := 0;
	    
	    "DBParAssi".MS.IN.Exe_MC_MoveRelative := FALSE;
	    "DBParAssi".MS.IN.Exe_MC_MoveAbs := FALSE;
	    "DBParAssi".MS.IN.Exe_MC_Halt := FALSE;
	    "FB_RIPRISTINO_MS_DB".fase := 0;
	    "FB_RIPRISTINO_MS_DB".bStart := 0;
	    "FB_RIPRISTINO_MS_DB".bDone := 0;
	    
	    "DBParAssi".ME.IN.Exe_MC_MoveRelative := FALSE;
	    "DBParAssi".ME.IN.Exe_MC_MoveAbs := FALSE;
	    "DBParAssi".ME.IN.Exe_MC_Halt := FALSE;
	    "FB_RIPRISTINO_ME_DB".bStart := 0;
	    "FB_RIPRISTINO_ME_DB".fase := 0;
	    "FB_RIPRISTINO_ME_DB".bDone := 0;
	    
	    // Reset seq
	    // 
	    "FB_CICLO_DB".fase := 0;
	    "STARTCICLO" := 0;
	    "RIPRISTINO" := 0;
	    "FB_RIPRISTINO_GEN_DB".fase := 0;
	    "FB_RIPRISTINO_GEN_DB".bStart := 0;
	    
	    // varie
	    // 
	    "FB_CICLO_DB".appComandoIndietroME := FALSE;
	    
	    
	END_IF;
	
	
	
	
END_FUNCTION

FUNCTION_BLOCK "FB_CICLO_GEN_1"
{ S7_Optimized_Access := 'TRUE' }
VERSION : 0.1
   VAR_OUTPUT 
      fase : Int := 0;   // fase attiva
   END_VAR

   VAR 
      condOkStartCiclo { S7_SetPoint := 'True'} : Bool;
      T10 {InstructionName := 'TON_TIME'; LibVersion := '1.0'} : TON_TIME;
      T20 {InstructionName := 'TON_TIME'; LibVersion := '1.0'} : TON_TIME;
      T30 {InstructionName := 'TON_TIME'; LibVersion := '1.0'} : TON_TIME;
      T40 {InstructionName := 'TON_TIME'; LibVersion := '1.0'} : TON_TIME;
      T50 {InstructionName := 'TON_TIME'; LibVersion := '1.0'} : TON_TIME;
      T60 {InstructionName := 'TON_TIME'; LibVersion := '1.0'} : TON_TIME;
      T70 {InstructionName := 'TON_TIME'; LibVersion := '1.0'} : TON_TIME;
      T75 {InstructionName := 'TON_TIME'; LibVersion := '1.0'} : TON_TIME;
      T80 {InstructionName := 'TON_TIME'; LibVersion := '1.0'} : TON_TIME;
      T90 {InstructionName := 'TON_TIME'; LibVersion := '1.0'} : TON_TIME;
      T100 {InstructionName := 'TON_TIME'; LibVersion := '1.0'} : TON_TIME;
      TcicloPrec { S7_SetPoint := 'True'} : Int;
      TCicloAtt : Int;
      appQuotaStartStrappi : Real;
      FNStartCiclo : Bool;
      AppFNStartCiclo : Bool;
      FPClok01s : Bool;
      AppFPClok01s : Bool;
      appComandoIndietroME : Bool;
   END_VAR

   VAR CONSTANT 
      T_DELAY_SEQ : Time;
      T_DELAY_SCANSIONE : Time := T#20ms;
   END_VAR


BEGIN
	// ciclo generale
	// v0.1 passo passo
	// v0.2 calcolo quota
	// v0.3 indetro ME su quota strappi
	REGION Timers
	    
	    #T10(IN := #fase = 10,
	         PT := #T_DELAY_SEQ);
	    
	    #T20(IN := #fase = 20,
	         PT := #T_DELAY_SEQ);
	    
	    #T30(IN := #fase = 30,
	         PT := #T_DELAY_SEQ);
	    
	    #T40(IN := #fase = 40,
	         PT := #T_DELAY_SEQ);
	    
	    #T50(IN := #fase = 50,
	         PT := #T_DELAY_SEQ);
	    
	    #T60(IN := #fase = 60,
	         PT := #T_DELAY_SEQ);
	    
	    #T70(IN := #fase = 70,
	         PT := #T_DELAY_SCANSIONE);
	    
	    #T80(IN := #fase = 80,
	         PT := #T_DELAY_SEQ);
	    
	    #T75(IN := #fase = 75,
	         PT := #T_DELAY_SEQ);
	    
	    #T90(IN := #fase = 90,
	         PT := #T_DELAY_SCANSIONE);
	    
	    #T100(IN := #fase = 100,
	          PT := #T_DELAY_SEQ);
	END_REGION
	
	// CONDIZIONI 
	// 
	#condOkStartCiclo := "AUTOMATICO" AND "RIPRISTINATO" AND "AUX_OK_T";
	
	// reset start
	// 
	IF NOT #condOkStartCiclo THEN
	    "STARTCICLO" := FALSE;
	END_IF;
	
	CASE #fase OF
	        
	    0: // introduzione MA + ME insieme + MS quota MA
	        IF "STARTCICLO" AND #condOkStartCiclo THEN
	            IF "PASSO_PASSO" THEN
	                "STARTCICLO" := FALSE;
	            END_IF;
	            // comandi
	            // MA
	            "DBParAssi".MA.IN.Sp_MoveAbs_Position := "DBParAssi".MA.pos."1"; // 7.5 mm
	            "DBParAssi".MA.IN.Exe_MC_MoveAbs := TRUE;
	            // ME
	            "DBParAssi".ME.IN.Sp_MoveAbs_Position := "DBParAssi".ME.pos."1"; // 120°
	            "DBParAssi".ME.IN.Exe_MC_MoveAbs := TRUE;
	            // MS
	            "DBParAssi".MS.IN.Sp_MoveRel_Distance := "DBParAssi".MS.pos."3"; // quota MA
	            "DBParAssi".MS.IN.Sp_MoveRel_Velocity := "DBParAssi".MS.vel."3"; // velocita
	            "DBParAssi".MS.IN.Exe_MC_MoveRelative := TRUE;
	            
	            #fase := 10;
	        END_IF;
	        
	    10: // detorsione
	        IF #T10.Q
	            AND "STARTCICLO"
	            AND "DBParAssi".MA.OUT.Output_MC_MoveAbs_Done
	            AND "DBParAssi".ME.OUT.Output_MC_MoveAbs_Done
	            AND "DBParAssi".MS.OUT.Output_MC_MoveRel_Done
	        THEN
	            IF "PASSO_PASSO" THEN
	                "STARTCICLO" := FALSE;
	            END_IF;
	            // comandi
	            // MA
	            "DBParAssi".MA.IN.Exe_MC_MoveAbs := FALSE;
	            // MS
	            "DBParAssi".MS.IN.Exe_MC_MoveRelative := FALSE;
	            // ME
	            "DBParAssi".ME.IN.Exe_MC_MoveAbs := FALSE;
	            // MR
	            "DBParAssi".MR.IN.Sp_MoveAbs_Position := "DBParAssi".MR.pos."2"; // X° quota intermedia detorsione parziale
	            "DBParAssi".MR.IN.Sp_MoveAbs_Velocity := "DBParAssi".MR.vel."2";
	            "DBParAssi".MR.IN.Exe_MC_MoveAbs := TRUE;
	            
	            #fase := 20;
	        END_IF;
	        
	    20: // ME -
	        IF #T20.Q
	            AND "STARTCICLO"
	            AND "DBParAssi".MR.OUT.Output_MC_MoveAbs_Done
	        THEN
	            // IF "PASSO_PASSO" THEN
	            //     "STARTCICLO" := FALSE;
	            // END_IF;
	            // comandi
	            // MR
	            "DBParAssi".MR.IN.Exe_MC_MoveAbs := FALSE;
	            // ME
	            "DBParAssi".ME.IN.Sp_MoveAbs_Position := "DBParAssi".ME.pos."2"; // 0°
	            "DBParAssi".ME.IN.Exe_MC_MoveAbs := TRUE;
	            
	            #fase := 30;
	        END_IF;
	        
	    30:  // avanti MA
	        IF #T30.Q AND "STARTCICLO"
	            AND "DBParAssi"."ME".OUT.Output_MC_MoveAbs_Done
	        THEN
	            IF "PASSO_PASSO" THEN
	                "STARTCICLO" := FALSE;
	            END_IF;
	            // comandi
	            // ME
	            "DBParAssi".ME.IN.Exe_MC_MoveAbs := FALSE;
	            // MA
	            "DBParAssi".MA.IN.Sp_MoveAbs_Position := "DBParAssi".MA.pos."2"; // 12.5 mm
	            "DBParAssi".MA.IN.Exe_MC_MoveAbs := TRUE;
	            
	            #fase := 40;
	        END_IF;
	        
	    40: // avanti MS
	        IF #T40.Q
	            AND "STARTCICLO"
	            AND "DBParAssi".MA.OUT.Output_MC_MoveAbs_Done
	        THEN
	            IF "PASSO_PASSO" THEN
	                "STARTCICLO" := FALSE;
	            END_IF;
	            // comandi
	            // MA
	            "DBParAssi".MA.IN.Exe_MC_MoveAbs := FALSE;
	            // MS  
	            // "DBParAssi".MS.IN.Sp_MoveRel_Distance := "DBParAssi".MS.pos."2";
	            "DBParAssi".MS.IN.Sp_MoveRel_Distance := 800.0 - "DBParAssi".MS.pos."3"; // calcolo in base a quota MA
	            "DBParAssi".MS.IN.Exe_MC_MoveRelative := TRUE;
	            // // ME
	            // "DBParAssi".ME.IN.Sp_MoveAbs_Position := "DBParAssi".ME.pos."2"; // 0°
	            // "DBParAssi".ME.IN.Exe_MC_MoveAbs := TRUE;
	            
	            // staticizzo quota partenza Strappi
	            // 
	            #appQuotaStartStrappi := "DBParAssi".MS.OUT.Output_ActPos;
	            #appComandoIndietroME := TRUE;
	            
	            #fase := 50;
	        END_IF;
	        
	    50:   // fine detorsione MA
	        IF #T50.Q
	            AND "STARTCICLO"
	            AND "DBParAssi".MS.OUT.Output_MC_MoveRel_Done
	            // AND "DBParAssi"."ME".OUT.Output_MC_MoveAbs_Done
	        THEN
	            IF "PASSO_PASSO" THEN
	                "STARTCICLO" := FALSE;
	            END_IF;
	            // comandi
	            // MS
	            "DBParAssi".MS.IN.Exe_MC_MoveRelative := FALSE;
	            // // ME
	            // "DBParAssi".ME.IN.Exe_MC_MoveAbs := FALSE;
	            // MA indietro
	            "DBParAssi".MA.IN.Sp_MoveAbs_Position := "DBParAssi".MA.pos."1"; // 7.5 mm
	            "DBParAssi".MA.IN.Exe_MC_MoveAbs := TRUE;
	            
	            #fase := 55;
	        END_IF;
	        
	    55: // MR indietro per ritorsione
	        IF "STARTCICLO"
	            AND "DBParAssi".MA.OUT.Output_MC_MoveAbs_Done
	        THEN
	            IF "PASSO_PASSO" THEN
	                "STARTCICLO" := FALSE;
	            END_IF;
	            // comandi
	            // MA
	            "DBParAssi".MA.IN.Exe_MC_MoveAbs := FALSE;
	            // MR indietro
	            "DBParAssi".MR.IN.Sp_MoveAbs_Position := "DBParAssi".MR.pos."3"; // 0°
	            "DBParAssi".MR.IN.Sp_MoveAbs_Velocity := "DBParAssi".MR.vel."3";
	            "DBParAssi".MR.IN.Exe_MC_MoveAbs := TRUE;
	            
	            #fase := 60;
	        END_IF;
	        
	    60: // attesa ritosione MR indietro
	        IF #T60.Q
	            AND "STARTCICLO"
	            AND "DBParAssi".MR.OUT.Output_MC_MoveAbs_Done
	        THEN
	            // IF "PASSO_PASSO" THEN
	            //     "STARTCICLO" := FALSE;
	            // END_IF;
	            // comandi
	            // MR
	            "DBParAssi".MR.IN.Exe_MC_MoveAbs := FALSE;
	            
	            #fase := 70;
	        END_IF;
	        
	    70:// ritorsione  MA a 9.6mm
	        IF #T70.Q
	            AND "STARTCICLO"
	        THEN
	            IF "PASSO_PASSO" THEN
	                "STARTCICLO" := FALSE;
	            END_IF;
	            // comandi
	            // MA
	            "DBParAssi".MA.IN.Sp_MoveAbs_Position := "DBParAssi".MA.pos."3"; // 9.6 mm
	            "DBParAssi".MA.IN.Exe_MC_MoveAbs := TRUE;
	            
	            #fase := 75;
	        END_IF;
	        
	    75:// ritorsione MR a 80°
	        IF #T75.Q
	            AND "STARTCICLO"
	            AND "DBParAssi".MA.OUT.Output_MC_MoveAbs_Done
	        THEN
	            IF "PASSO_PASSO" THEN
	                "STARTCICLO" := FALSE;
	            END_IF;
	            // comandi
	            // MA
	            "DBParAssi".MA.IN.Exe_MC_MoveAbs := FALSE;
	            // MR
	            "DBParAssi".MR.IN.Sp_MoveAbs_Position := "DBParAssi".MR.pos."4"; // 80°
	            "DBParAssi".MR.IN.Sp_MoveAbs_Velocity := "DBParAssi".MR.vel."4";
	            "DBParAssi".MR.IN.Exe_MC_MoveAbs := TRUE;
	            
	            #fase := 80;
	        END_IF;
	        
	    80: // attesa segnali
	        IF #T80.Q
	            AND "STARTCICLO"
	            AND "DBParAssi".MR.OUT.Output_MC_MoveAbs_Done
	        THEN
	            // IF "PASSO_PASSO" THEN
	            //     "STARTCICLO" := FALSE;
	            // END_IF;
	            // comandi
	            // MR
	            "DBParAssi".MR.IN.Exe_MC_MoveAbs := FALSE;
	            
	            #fase := 90;
	        END_IF;
	        
	    90: //  fineciclo MA a 0mm  
	        IF #T90.Q
	            AND "STARTCICLO"
	        THEN
	            IF "PASSO_PASSO" THEN
	                "STARTCICLO" := FALSE;
	            END_IF;
	            // comandi
	            // MA
	            "DBParAssi".MA.IN.Sp_MoveAbs_Position := "DBParAssi".MA.pos."4"; // 0.0 mm
	            "DBParAssi".MA.IN.Exe_MC_MoveAbs := TRUE;
	            
	            #fase := 100;
	        END_IF;
	        
	    100:// MR ritorna a pos 1
	        IF #T100.Q
	            AND "STARTCICLO"
	            AND "DBParAssi".MA.OUT.Output_MC_MoveAbs_Done
	        THEN
	            IF "PASSO_PASSO" THEN
	                "STARTCICLO" := FALSE;
	            END_IF;
	            // comandi
	            // MA
	            "DBParAssi".MA.IN.Exe_MC_MoveAbs := FALSE;
	            // MR
	            "DBParAssi".MR.IN.Sp_MoveAbs_Position := "DBParAssi".MR.pos."1";
	            "DBParAssi".MR.IN.Sp_MoveAbs_Velocity := "DBParAssi".MR.vel."1";
	            "DBParAssi".MR.IN.Exe_MC_MoveAbs := TRUE;
	            
	            #fase := 200;
	        END_IF;
	        
	    200: // fineciclo
	        IF "DBParAssi".MR.OUT.Output_MC_MoveAbs_Done THEN
	            // comandi
	            // MA
	            "DBParAssi".MR.IN.Exe_MC_MoveAbs := FALSE;
	            "STARTCICLO" := FALSE;
	            
	            #fase := 0;
	        END_IF;
	        
	END_CASE;
	
	REGION Indietro ME a quota
	    // passo parallelo indietro ME risp quota MS
	    // i blocchi vanno indietro quando raggiungo la quota desiderata
	    IF #appComandoIndietroME AND ("DBParAssi".MS.OUT.Output_ActPos >= #appQuotaStartStrappi + 0.0) THEN  // era +10.0
	        // ME indietro
	        // "DBParAssi".ME.IN.Sp_MoveAbs_Position := "DBParAssi".ME.pos."2"; // 0°
	        // "DBParAssi".ME.IN.Exe_MC_MoveAbs := TRUE;
	        // azzero passo appoggio 
	        // 
	        #appComandoIndietroME := FALSE;
	    END_IF;
	    
	END_REGION
	
	REGION T ciclo
	    // tempo ciclo
	    // 
	    
	    // clock
	    // 
	    #FPClok01s := "Clock_10Hz" AND NOT #AppFPClok01s;
	    #AppFPClok01s := "Clock_10Hz";
	    
	    #FNStartCiclo := NOT "STARTCICLO" AND NOT #AppFNStartCiclo;
	    #AppFNStartCiclo := NOT "STARTCICLO";
	    
	    IF "STARTCICLO" AND #FPClok01s THEN
	        #TCicloAtt := #TCicloAtt + 1;
	    END_IF;
	    
	    // staticizzo
	    // 
	    IF #FNStartCiclo THEN
	        #TcicloPrec := #TCicloAtt;
	        #TCicloAtt := 0;
	    END_IF;
	    
	END_REGION
	
	
END_FUNCTION_BLOCK

FUNCTION_BLOCK "FB_RIPRISTINO_MR_1"
{ S7_Optimized_Access := 'TRUE' }
VERSION : 0.1
   VAR_OUTPUT 
      bDone : Bool;   // fine ciclo
      fase : Int;
   END_VAR

   VAR_IN_OUT 
      bStart : Bool;   // start ciclo
   END_VAR

   VAR 
      T20 {InstructionName := 'TON_TIME'; LibVersion := '1.0'; S7_SetPoint := 'False'} : TON_TIME;
   END_VAR


BEGIN
	// ripristino MR
	// 
	
	#T20(IN:=#fase = 20,
	     PT:=t#1s);
	
	CASE #fase OF
	        
	    0:// attendo start
	        IF #bStart THEN
	            // comandi
	            #bDone := FALSE;
	            "DBParAssi".MR.IN.Exe_MC_Home := FALSE; // resetto homed
	            "DBParAssi".MR.IN.Sp_MoveRel_Distance := -200.0;// vado indietro di x° era 200
	            "DBParAssi".MR.IN.Sp_MoveAbs_Velocity := "DBParAssi".MR.vel."1";
	            "DBParAssi".MR.IN.Exe_MC_MoveRelative := TRUE;
	            
	            #fase := 10;
	        END_IF;
	        
	    10:
	        IF "DBParAssi".MR.OUT.Output_MC_MoveRel_Done THEN
	            // comandi
	            "DBParAssi".MR.IN.Exe_MC_MoveRelative := FALSE;
	            "DBParAssi".MR.IN.Exe_MC_Home := TRUE;// azzero quota
	            
	            #fase := 20;
	        END_IF;
	        
	    20:
	        IF "DBParAssi".MR.OUT.Output_MC_AxisHomed AND #T20.Q THEN
	            // comandi
	            //"DBParAssi".MR.IN.Exe_MC_Home := FALSE;
	            "DBParAssi".MR.IN.Sp_MoveAbs_Position := "DBParAssi".MR.pos."1";// preset posizione 
	            "DBParAssi".MR.IN.Sp_MoveAbs_Velocity := "DBParAssi".MR.vel."1";
	            "DBParAssi".MR.IN.Exe_MC_MoveAbs := TRUE;
	            
	            #fase := 30;
	        END_IF;
	        
	    30:// fineciclo
	        IF "DBParAssi".MR.OUT.Output_MC_MoveAbs_Done THEN
	            // comandi
	            "DBParAssi".MR.IN.Exe_MC_MoveAbs := FALSE;
	            #bDone := TRUE;
	            #bStart := FALSE;
	            #fase := 0;
	        END_IF;
	        
	END_CASE;
	
	
	
	
	
END_FUNCTION_BLOCK

FUNCTION_BLOCK "FB_RIPRISTINO_MS_1"
{ S7_Optimized_Access := 'TRUE' }
VERSION : 0.1
   VAR_OUTPUT 
      bDone : Bool;   // fine ciclo
      fase : Int;
   END_VAR

   VAR_IN_OUT 
      bStart : Bool;   // start ciclo
   END_VAR

   VAR 
      T0 {InstructionName := 'TON_TIME'; LibVersion := '1.0'; S7_SetPoint := 'False'} : TON_TIME;
      T35 {InstructionName := 'TON_TIME'; LibVersion := '1.0'; S7_SetPoint := 'False'} : TON_TIME;
   END_VAR


BEGIN
	// ripristino MS (gestito unita' di mis ad impulsi 400 impulsi / giro) rapporto di rid 1/2
	// 
	
	// #T20(IN:=#fase = 20,
	//      PT:=t#1s);
	
	#T0(IN := #bStart,
	     PT := t#20Ms);
	 
	#T35(IN := #fase = 35,
	     PT := t#0.5s);
	
	CASE #fase OF
	        
	    0:// attendo start
	        IF #bStart THEN
	            // comandi
	            #bDone := FALSE;
	            "DBParAssi".MS.IN.Exe_MC_Home := FALSE; // resetto homed
	            "DBParAssi".MS.IN.Sp_MoveRel_Distance := 800;// mando avanti di x [pulses] fino che prendo il sensore 800 = 2 giri
	            "DBParAssi".MS.IN.Exe_MC_MoveRelative := TRUE;
	            "DBParAssi".MS.IN.Sp_MoveRel_Velocity := 500; // p/s vel ripristino
	            
	            #fase := 10;
	        END_IF;
	        
	    10:
	        IF "DBParAssi".MS.OUT.Output_MC_MoveRel_Done OR "E0.0 FC HOMING MS"  THEN  // qui fare allarme no homing
	            IF NOT "E0.0 FC HOMING MS" THEN
	                "ALLA_01_FC_HOMING_MS" := TRUE;
	                #fase := 900;  // fineciclo con allarme
	            ELSE
	                // comandi
	                "DBParAssi".MS.IN.Exe_MC_Halt := TRUE;
	                "DBParAssi".MS.IN.Exe_MC_MoveRelative := FALSE;
	                "DBParAssi".MS.IN.Sp_MoveRel_Velocity := 1000; // p/s vel ripristino
	              
	                #fase := 20;
	            END_IF;
	        END_IF;
	        
	    20:
	        IF "DBParAssi".MS.OUT.Output_MC_Halt_Done  THEN
	            // comandi
	            // 
	            "DBParAssi".MS.IN.Exe_MC_Home := TRUE;// azzero quota
	            
	            #fase := 35;
	        END_IF;
	        
	    35:
	        IF "DBParAssi".MS.OUT.Output_MC_AxisHomed AND #T35.Q THEN
	            // comandi
	            // 
	            "DBParAssi".MS.IN.Exe_MC_Halt := FALSE;
	            "DBParAssi".MS.IN.Sp_MoveRel_Distance := "DBParAssi".MS.pos."1";// preset posizione per partenza
	            "DBParAssi".MS.IN.Exe_MC_MoveRelative := TRUE;
	            
	            #fase := 40;
	        END_IF;
	        
	    40:// fineciclo
	        IF TRUE THEN
	            // comandi
	            "DBParAssi".MS.IN.Exe_MC_MoveRelative := FALSE;
	            #bDone := TRUE;
	            #bStart := FALSE;
	            
	            #fase := 0;
	        END_IF;
	        
	    900:// fineciclo x allarme
	        // comandi
	        // 
	        "DBParAssi".MS.IN.Exe_MC_MoveRelative := FALSE;
	        #bStart := FALSE;
	        
	END_CASE;
	
	
	
	
	
END_FUNCTION_BLOCK

DATA_BLOCK "FB_STATI_MACCHINA_DB"   // DB9
VERSION : 0.1
// stored: AutoNumber true, DBAccessibleFromOPCUA true, InstanceOfName FB_STATI_MACCHINA, InstanceOfType FB
"FB_STATI_MACCHINA"
BEGIN
END_DATA_BLOCK

DATA_BLOCK "CTRL_ASSE_DB"   // DB4
VERSION : 0.1
// stored: AutoNumber true, DBAccessibleFromOPCUA true, InstanceOfName CTRL_ASSE_STD, InstanceOfType FB
"CTRL_ASSE_STD"
   // VAR_INPUT
   //    Automatico : Bool;
   //    Exe_MC_Reset : Bool;
   //    En_MC_Power : Bool;
   //    Exe_MC_Home : Bool;
   //    Sp_Offset_Homing : Real;
   //    Sp_Homing_Mode : Int;
   //    Exe_MC_Halt : Bool;
   //    Exe_Jog_Fwd : Bool;
   //    Exe_Jog_Bkw : Bool;
   //    Sp_Jog_Velocity : Real;
   //    Exe_MC_Velocity : Bool;
   //    Sp_MC_Velocity : Real;
   //    Exe_MC_Relative : Bool;
   //    Sp_MoveRel_Distance : Real;
   //    Sp_MoveRel_Velocity : Real;
   //    Exe_MC_Abs : Bool;
   //    Sp_MoveAbs_Position : Real;
   //    Sp_MoveAbs_Velocity : Real;
   //    Exe_MC_ChangeDyna : Bool;
   //    Sp_RampUpTime : Real;
   //    Sp_RampDnTime : Real;
   // END_VAR
   // VAR_OUTPUT
   //    Output_MC_Reset_Done : Bool;
   //    Output_MC_AxisEnabled : Bool;
   //    Output_MC_AxisHomed : Bool;
   //    Output_MC_Halt_Done : Bool;
   //    Output_MC_JogInVelocity : Bool;
   //    Output_MC_MoveInVelocity : Bool;
   //    Output_MC_MoveRel_Done : Bool;
   //    Output_MC_MoveAbs_Done : Bool;
   //    Output_MC_MoveAbs_Busy : Bool;
   //    Output_MC_At_Standstill : Bool;
   //    Output_MC_Error : Bool;
   //    Output_ActVelocity : Real;
   //    Output_ActPos : Real;
   // END_VAR
   // VAR_IN_OUT
   //    AxisTO : TO_PositioningAxis;
   // END_VAR
   // VAR
   //    AxisReady_PosAxis { S7_SetPoint := 'True'} : Bool;
   //    MC_Power_Instance { S7_SetPoint := 'True'} : MC_Power;
   //    MC_Reset_Instance { S7_SetPoint := 'True'} : MC_Reset;
   //    MC_Halt_Instance { S7_SetPoint := 'True'} : MC_Halt;
   //    MC_MoveJog_Instance { S7_SetPoint := 'True'} : MC_MoveJog;
   //    MC_MoveAbsolute_Instance { S7_SetPoint := 'True'} : MC_MoveAbsolute;
   //    MC_MoveVelocity_Instance { S7_SetPoint := 'True'} : MC_MoveVelocity;
   //    MC_Home_Instance { S7_SetPoint := 'True'} : MC_Home;
   //    MC_MoveRelative_Instance { S7_SetPoint := 'True'} : MC_MoveRelative;
   //    MC_ChangeDynamic_Instance { S7_SetPoint := 'True'} : MC_ChangeDynamic;
   // END_VAR
BEGIN
END_DATA_BLOCK

DATA_BLOCK "CTRL_ASSE_STD_DB_MR"   // DB7
VERSION : 0.1
// stored: AutoNumber true, DBAccessibleFromOPCUA true, InstanceOfName CTRL_ASSE_STD, InstanceOfType FB
"CTRL_ASSE_STD"
   // VAR_INPUT
   //    Automatico : Bool;
   //    Exe_MC_Reset : Bool;
   //    En_MC_Power : Bool;
   //    Exe_MC_Home : Bool;
   //    Sp_Offset_Homing : Real;
   //    Sp_Homing_Mode : Int;
   //    Exe_MC_Halt : Bool;
   //    Exe_Jog_Fwd : Bool;
   //    Exe_Jog_Bkw : Bool;
   //    Sp_Jog_Velocity : Real;
   //    Exe_MC_Velocity : Bool;
   //    Sp_MC_Velocity : Real;
   //    Exe_MC_Relative : Bool;
   //    Sp_MoveRel_Distance : Real;
   //    Sp_MoveRel_Velocity : Real;
   //    Exe_MC_Abs : Bool;
   //    Sp_MoveAbs_Position : Real;
   //    Sp_MoveAbs_Velocity : Real;
   //    Exe_MC_ChangeDyna : Bool;
   //    Sp_RampUpTime : Real;
   //    Sp_RampDnTime : Real;
   // END_VAR
   // VAR_OUTPUT
   //    Output_MC_Reset_Done : Bool;
   //    Output_MC_AxisEnabled : Bool;
   //    Output_MC_AxisHomed : Bool;
   //    Output_MC_Halt_Done : Bool;
   //    Output_MC_JogInVelocity : Bool;
   //    Output_MC_MoveInVelocity : Bool;
   //    Output_MC_MoveRel_Done : Bool;
   //    Output_MC_MoveAbs_Done : Bool;
   //    Output_MC_MoveAbs_Busy : Bool;
   //    Output_MC_At_Standstill : Bool;
   //    Output_MC_Error : Bool;
   //    Output_ActVelocity : Real;
   //    Output_ActPos : Real;
   // END_VAR
   // VAR_IN_OUT
   //    AxisTO : TO_PositioningAxis;
   // END_VAR
   // VAR
   //    AxisReady_PosAxis { S7_SetPoint := 'True'} : Bool;
   //    MC_Power_Instance { S7_SetPoint := 'True'} : MC_Power;
   //    MC_Reset_Instance { S7_SetPoint := 'True'} : MC_Reset;
   //    MC_Halt_Instance { S7_SetPoint := 'True'} : MC_Halt;
   //    MC_MoveJog_Instance { S7_SetPoint := 'True'} : MC_MoveJog;
   //    MC_MoveAbsolute_Instance { S7_SetPoint := 'True'} : MC_MoveAbsolute;
   //    MC_MoveVelocity_Instance { S7_SetPoint := 'True'} : MC_MoveVelocity;
   //    MC_Home_Instance { S7_SetPoint := 'True'} : MC_Home;
   //    MC_MoveRelative_Instance { S7_SetPoint := 'True'} : MC_MoveRelative;
   //    MC_ChangeDynamic_Instance { S7_SetPoint := 'True'} : MC_ChangeDynamic;
   // END_VAR
BEGIN
END_DATA_BLOCK

DATA_BLOCK "FB_ORG_ASSI_DB"   // DB13
VERSION : 0.1
// stored: AutoNumber true, DBAccessibleFromOPCUA true, InstanceOfName FB_ORG_ASSI, InstanceOfType FB
"FB_ORG_ASSI"
BEGIN
END_DATA_BLOCK

DATA_BLOCK "FB_PosizAsseStandard_DB"   // DB5
VERSION : 0.1
// stored: AutoNumber true, DBAccessibleFromOPCUA true, InstanceOfName FB_PosizAsseStandard, InstanceOfType FB
"FB_PosizAsseStandard"
   // VAR_INPUT
   //    Exe_MC_Reset : Bool;
   //    En_MC_Power : Bool;
   //    Exe_MC_Home : Bool;
   //    Exe_Jog_Fwd : Bool;
   //    Exe_Jog_Rev : Bool;
   //    Exe_MC_Velocity : Bool;
   //    Exe_MC_Relative : Bool;
   //    Exe_MC_Abs : Bool;
   //    Exe_MC_Halt : Bool;
   //    Ctl_MC_Stop : Bool;
   //    Sp_lr_MC_HomingOffset : LReal;
   //    Sp_lr_MC_Velocity : LReal;
   //    Sp_lr_MC_RelativeDistance : LReal;
   //    Sp_lr_MC_AbsPosition : LReal;
   // END_VAR
   // VAR_OUTPUT
   //    Output_MC_At_Standstill : Bool;
   //    Output_MC_AxisEnabled : Bool;
   //    Output_MC_MoveAbs_Done : Bool;
   //    Output_MC_MoveAbs_Busy : Bool;
   //    Output_MC_Error : Bool;
   //    Output_MC_AxisHomed : Bool;
   //    Output_ActVelocity : Real;
   //    Output_ActPos : Real;
   // END_VAR
   // VAR_IN_OUT
   //    AxisTO : TO_PositioningAxis;
   // END_VAR
   // VAR
   //    AxisReady_PosAxis { S7_SetPoint := 'True'} : Bool;
   //    MC_Power_Instance_1 { S7_SetPoint := 'True'} : MC_Power;
   //    MC_Home_Instance_1 { S7_SetPoint := 'True'} : MC_Home;
   //    MC_MoveJog_Instance_1 { S7_SetPoint := 'True'} : MC_MoveJog;
   //    MC_MoveVelocity_Instance_1 { S7_SetPoint := 'True'} : MC_MoveVelocity;
   //    MC_MoveRelative_Instance_1 { S7_SetPoint := 'True'} : MC_MoveRelative;
   //    MC_MoveAbsolute_Instance_1 { S7_SetPoint := 'True'} : MC_MoveAbsolute;
   //    MC_Halt_Instance_1 { S7_SetPoint := 'True'} : MC_Halt;
   //    MC_Reset_Instance_1 { S7_SetPoint := 'True'} : MC_Reset;
   // END_VAR
BEGIN
END_DATA_BLOCK

DATA_BLOCK "FB_CICLO_DB"   // DB11
VERSION : 0.1
// stored: AutoNumber true, DBAccessibleFromOPCUA true, InstanceOfName FB_CICLO_GEN, InstanceOfType FB
"FB_CICLO_GEN"
   // VAR_OUTPUT
   //    fase : Int;
   // END_VAR
   // VAR
   //    condOkStartCiclo { S7_SetPoint := 'True'} : Bool;
   //    T10 { S7_SetPoint := 'True'} : TON_TIME;
   //    T20 { S7_SetPoint := 'True'} : TON_TIME;
   //    T30 { S7_SetPoint := 'True'} : TON_TIME;
   //    T40 { S7_SetPoint := 'True'} : TON_TIME;
   //    T50 { S7_SetPoint := 'True'} : TON_TIME;
   //    T60 { S7_SetPoint := 'True'} : TON_TIME;
   //    T70 { S7_SetPoint := 'True'} : TON_TIME;
   //    T75 { S7_SetPoint := 'True'} : TON_TIME;
   //    T80 { S7_SetPoint := 'True'} : TON_TIME;
   //    T90 { S7_SetPoint := 'True'} : TON_TIME;
   //    T100 { S7_SetPoint := 'True'} : TON_TIME;
   //    TcicloPrec { S7_SetPoint := 'True'} : Int;
   //    TCicloAtt : Int;
   //    appQuotaStartStrappi : Real;
   //    FNStartCiclo : Bool;
   //    AppFNStartCiclo : Bool;
   //    FPClok01s : Bool;
   //    AppFPClok01s : Bool;
   //    appComandoIndietroME : Bool;
   // END_VAR
BEGIN
END_DATA_BLOCK

DATA_BLOCK "FB_RIPRISTINO_GEN_DB"   // DB10
VERSION : 0.1
// stored: AutoNumber true, DBAccessibleFromOPCUA true, InstanceOfName FB_RIPRISTINO_GEN, InstanceOfType FB
"FB_RIPRISTINO_GEN"
BEGIN
END_DATA_BLOCK

DATA_BLOCK "FB_RIPRISTINO_MA_DB"   // DB15
VERSION : 0.1
// stored: AutoNumber true, DBAccessibleFromOPCUA true, InstanceOfName FB_RIPRISTINO_MA, InstanceOfType FB
"FB_RIPRISTINO_MA"
   // VAR_OUTPUT
   //    bDone : Bool;
   //    fase : Int;
   // END_VAR
   // VAR_IN_OUT
   //    bStart : Bool;
   // END_VAR
   // VAR
   //    T20 : TON_TIME;
   // END_VAR
BEGIN
END_DATA_BLOCK

DATA_BLOCK "FB_RIPRISTINO_ME_DB"   // DB17
VERSION : 0.1
// stored: AutoNumber true, DBAccessibleFromOPCUA true, InstanceOfName FB_RIPRISTINO_ME, InstanceOfType FB
"FB_RIPRISTINO_ME"
   // VAR_OUTPUT
   //    bDone : Bool;
   //    fase : Int;
   // END_VAR
   // VAR_IN_OUT
   //    bStart : Bool;
   // END_VAR
   // VAR
   //    T20 : TON_TIME;
   // END_VAR
BEGIN
END_DATA_BLOCK

DATA_BLOCK "FB_RIPRISTINO_MR_DB"   // DB14
VERSION : 0.1
// stored: AutoNumber true, DBAccessibleFromOPCUA true, InstanceOfName FB_RIPRISTINO_MR, InstanceOfType FB
"FB_RIPRISTINO_MR"
   // VAR_OUTPUT
   //    bDone : Bool;
   //    fase : Int;
   // END_VAR
   // VAR_IN_OUT
   //    bStart : Bool;
   // END_VAR
   // VAR
   //    T10 : TON_TIME;
   //    T20 : TON_TIME;
   // END_VAR
BEGIN
END_DATA_BLOCK

DATA_BLOCK "FB_RIPRISTINO_MS_DB"   // DB16
VERSION : 0.1
// stored: AutoNumber true, DBAccessibleFromOPCUA true, InstanceOfName FB_RIPRISTINO_MS, InstanceOfType FB
"FB_RIPRISTINO_MS"
   // VAR_OUTPUT
   //    bDone : Bool;
   //    fase : Int;
   // END_VAR
   // VAR_IN_OUT
   //    bStart : Bool;
   // END_VAR
   // VAR
   //    T10 : TON_TIME;
   //    T35 : TON_TIME;
   // END_VAR
BEGIN
END_DATA_BLOCK

DATA_BLOCK "ALLARMI_DB"   // DB19
VERSION : 0.1
// stored: AutoNumber true, DBAccessibleFromOPCUA true, InstanceOfName ALLARMI, InstanceOfType FB
"ALLARMI"
BEGIN
END_DATA_BLOCK
